(* Logix 5000 project; controller PHOTON Emulate 5570 rev 30.12; software revision 30.00 *)

TASK MainTask (periodic, rate 10000 ms, priority 1, watchdog 10000 ms) : MainProgram

MODULES
   Local : Emulate 5570 (ICP 2, rev 30.12)
       : vendor 1 type 0 code 15 (ICP 0, rev 1.1, Output RPI 50 ms)
END_MODULES

TYPE UDT_BA :
STRUCT
   AL : BOOL[128];
END_STRUCT
END_TYPE

VAR_GLOBAL   (* controller tags *)
   hash_valid : BOOL;
   hash_value : INT[32];
   hash_value_id : DINT;
   open_msg : INT[96];
   open_msg_id : DINT;
   open_msg_valid : BOOL;
   SCAN_CYCLE_TIME : DINT;
END_VAR

PROGRAM MainProgram   (* main routine MainRoutine *)
VAR
   PHT_Bit_indxj : DINT;
   PHT_Byte_indxi : DINT;
   PHT_Ceilmod : DINT;
   PHT_CeilRres : DINT;
   PHT_CompressFunction_BitOffSet : DINT;
   PHT_D : DINT;
   PHT_Digest : DINT[60];
   PHT_DIGESTSIZE : DINT;
   PHT_GetByte_BitOffSet : DINT;
   PHT_GetByte_i : DINT;
   PHT_GetByte_Indx : DINT;
   PHT_GetByte_j : DINT;
   PHT_GetByte_NoOfBits : DINT;
   PHT_GetByte_Res : DINT;
   PHT_hash_index : DINT;
   PHT_i : DINT;
   PHT_index : DINT;
   PHT_Init_i : DINT;
   PHT_isPadding : BOOL;
   PHT_IV : INT[8,8];
   PHT_j : DINT;
   PHT_Message : DINT[1024];
   PHT_MessIndex : DINT;
   PHT_MsgBitLen : DINT;
   PHT_Padded : DINT[1024];
   PHT_Padded_bound : DINT;
   PHT_Padded_Index : DINT;
   PHT_Per_i : DINT;
   PHT_Per_j : DINT;
   PHT_Per_r : DINT;
   PHT_RATE : DINT;
   PHT_RATEP : DINT;
   PHT_RC : DINT[8,12];
   PHT_round : DINT;
   PHT_S : DINT;
   PHT_SCS_c : DINT;
   PHT_SCS_i : DINT;
   PHT_SCS_index : DINT;
   PHT_SCS_indxi : DINT;
   PHT_SCS_j : DINT;
   PHT_SCS_OS : DINT[8,8];
   PHT_SCS_r : DINT;
   PHT_SCS_v : DINT[2];
   PHT_Squeeze_i : DINT;
   PHT_Squeeze_tmp : DINT;
   PHT_State : DINT[8,8];
   PHT_Table : DINT[8,256,2];
   PHT_Tmp : DINT[2];
   PHT_Ver : DINT;
   PHT_WordToByte_BitOffSet : DINT;
   PHT_WordToByte_i : DINT;
   PHT_WordToByte_indxi : DINT;
   PHT_WordToByte_indxj : DINT;
   PHT_WordToByte_j : DINT;
   PHT_WordToByte_NoOfBits : DINT;
   PHT_WordToByte_WordOffset : DINT;
   PHT_WordXorByte_BitOffSet : DINT;
   PHT_WordXorByte_i : DINT;
   PHT_WordXorByte_j : DINT;
   PHT_WordXorByte_NoOfBits : DINT;
   PHT_WordXorByte_Str : DINT[1024];
   PHT_WordXorByte_WordOffset : DINT;
   PHT_WriteByte_BitOffset : DINT;
   PHT_WriteByte_i : DINT;
   PHT_WriteByte_LocalFilter : DINT;
   PHT_WriteByte_NoOfBits : DINT;
   PHT_WriteByte_Value : DINT;
   Test_i : DINT;
END_VAR

ROUTINE MainRoutine   (* ladder *)
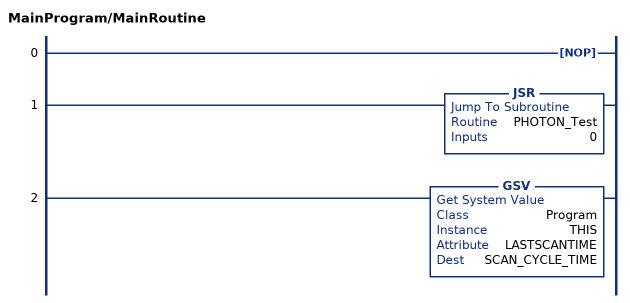
   0: NOP();
   1: JSR(PHOTON_Test,0);
   2: GSV(Program,THIS,LASTSCANTIME,SCAN_CYCLE_TIME);
END_ROUTINE

ROUTINE PHOTON   (* structured text *)
   
   
   JSR(PHOTON_Init);
   
   PHT_isPadding:=0;
   
   PHT_MessIndex:=0;
   while PHT_MessIndex <= PHT_MsgBitLen - PHT_RATE do
   
   	PHT_CompressFunction_BitOffSet:=PHT_MessIndex;
   	JSR(PHOTON_CompressFunction);
   
   	PHT_MessIndex:=PHT_MessIndex + PHT_RATE;
   end_while;
   
   
   PHT_Ceilmod:=PHT_MsgBitLen-PHT_MessIndex;
   PHT_Padded_bound:=PHT_Ceilmod/8;
   PHT_Ceilmod:= PHT_Ceilmod Mod 8;
   if PHT_Ceilmod<>0 then
   	PHT_Padded_bound:=PHT_Padded_bound+1;
   end_if;
   
   
   PHT_hash_index:=PHT_MessIndex/8;
   
   for PHT_i:=0 to PHT_Padded_bound-1 by 1 do
   	PHT_Padded[PHT_i]:=PHT_Message[PHT_hash_index + PHT_i];
   end_for;
   PHT_Padded[PHT_i]:=16#80;
   
   PHT_isPadding:=1;
   
   
   
   PHT_CompressFunction_BitOffSet:=PHT_MessIndex and 16#07;
   JSR(PHOTON_CompressFunction);
   
   
   JSR(PHOTON_Squeeze);
   
END_ROUTINE

ROUTINE PHOTON_CompressFunction   (* structured text *)
   
   PHT_WordXorByte_NoOfBits:=PHT_RATE;
   PHT_WordXorByte_WordOffset:=0;
   PHT_WordXorByte_BitOffSet:= PHT_CompressFunction_BitOffSet;
   
   JSR(PHOTON_WordXorByte);
   
   
   JSR(PHOTON_Permutation);
END_ROUTINE

ROUTINE PHOTON_GetByte   (* structured text *)
   (*byte GetByte(const byte*str, int BitOffSet, int NoOfBits)
       if S==8:
           if (BitOffSet & 0x7):
               res=((str[BitOffSet >> 3] << 4) | (str[(BitOffSet >> 3) + 1] >> 4))
           else:
               res=str[BitOffSet >> 3]
       else:
           res=(str[BitOffSet>>3] >> (4-(BitOffSet&0x4))) & ((1<<S)-1)
   
       return res
   	*)
   
   
   PHT_GetByte_Res:=0;
   
   PHT_GetByte_Indx:=PHT_GetByte_BitOffSet/8;
   
   If PHT_S=8 Then
   	PHT_Tmp[0]:=PHT_GetByte_BitOffSet AND 16#7;
   	if PHT_Tmp[0]<>0 Then
   		If PHT_isPadding Then
   			PHT_Tmp[0]:=PHT_Padded[PHT_GetByte_Indx]*16;
   			PHT_Tmp[1]:=PHT_Padded[PHT_GetByte_Indx+1]/16;
   		else
   			PHT_Tmp[0]:=PHT_Message[PHT_GetByte_Indx]*16;
   			PHT_Tmp[1]:=PHT_Message[PHT_GetByte_Indx+1]/16;
   		End_If;
   		PHT_GetByte_Res:=(PHT_Tmp[0] OR PHT_Tmp[1]) AND 16#FF;
   	else
   		If PHT_isPadding Then
   			PHT_GetByte_Res:=PHT_Padded[PHT_GetByte_Indx];
   		Else
   			PHT_GetByte_Res:=PHT_Message[PHT_GetByte_Indx];
   		End_If;
   	End_if;
   Else
   	If PHT_isPadding Then
   		PHT_Tmp[0]:=PHT_Padded[PHT_GetByte_Indx];
   	Else
   		PHT_Tmp[0]:=PHT_Message[PHT_GetByte_Indx];
   	End_If;
   
   
   	PHT_Tmp[1]:=4-(PHT_GetByte_BitOffSet AND 16#4);
   	Case PHT_Tmp[1] OF
   		1:
   			PHT_Tmp[0]:=PHT_Tmp[0]/2;
   		2:
   			PHT_Tmp[0]:=PHT_Tmp[0]/4;
   		3:
   			PHT_Tmp[0]:=PHT_Tmp[0]/8;
   		4:
   			PHT_Tmp[0]:=PHT_Tmp[0]/16;
   	End_CASE;
   	PHT_GetByte_Res:=PHT_Tmp[0] & 16#f;
   
   End_if;
   
   
END_ROUTINE

ROUTINE PHOTON_Init   (* structured text *)
   PHT_round:=12; // 12
   if PHT_Ver >= 5 then
   	PHT_S:= 8;
   else
   	PHT_S:=4;
   end_if;
   
   CASE PHT_Ver OF
   	 0:
   		PHT_D:=5;
   		PHT_S:=4;
   		PHT_RATE:=20;
   		PHT_RATEP:=16;
   		PHT_DIGESTSIZE:=80;
   		 PHT_RC[0,0]:=1;
   		 PHT_RC[0,1]:=3;
   		 PHT_RC[0,2]:=7;
   		 PHT_RC[0,3]:=14;
   		 PHT_RC[0,4]:=13;
   		 PHT_RC[0,5]:=11;
   		 PHT_RC[0,6]:=6;
   		 PHT_RC[0,7]:=12;
   		 PHT_RC[0,8]:=9;
   		 PHT_RC[0,9]:=2;
   		 PHT_RC[0,10]:=5;
   		 PHT_RC[0,11]:=10;
   		 PHT_RC[1,0]:=0;
   		 PHT_RC[1,1]:=2;
   		 PHT_RC[1,2]:=6;
   		 PHT_RC[1,3]:=15;
   		 PHT_RC[1,4]:=12;
   		 PHT_RC[1,5]:=10;
   		 PHT_RC[1,6]:=7;
   		 PHT_RC[1,7]:=13;
   		 PHT_RC[1,8]:=8;
   		 PHT_RC[1,9]:=3;
   		 PHT_RC[1,10]:=4;
   		 PHT_RC[1,11]:=11;
   		 PHT_RC[2,0]:=2;
   		 PHT_RC[2,1]:=0;
   		 PHT_RC[2,2]:=4;
   		 PHT_RC[2,3]:=13;
   		 PHT_RC[2,4]:=14;
   		 PHT_RC[2,5]:=8;
   		 PHT_RC[2,6]:=5;
   		 PHT_RC[2,7]:=15;
   		 PHT_RC[2,8]:=10;
   		 PHT_RC[2,9]:=1;
   		 PHT_RC[2,10]:=6;
   		 PHT_RC[2,11]:=9;
   		 PHT_RC[3,0]:=7;
   		 PHT_RC[3,1]:=5;
   		 PHT_RC[3,2]:=1;
   		 PHT_RC[3,3]:=8;
   		 PHT_RC[3,4]:=11;
   		 PHT_RC[3,5]:=13;
   		 PHT_RC[3,6]:=0;
   		 PHT_RC[3,7]:=10;
   		 PHT_RC[3,8]:=15;
   		 PHT_RC[3,9]:=4;
   		 PHT_RC[3,10]:=3;
   		 PHT_RC[3,11]:=12;
   		 PHT_RC[4,0]:=5;
   		 PHT_RC[4,1]:=7;
   		 PHT_RC[4,2]:=3;
   		 PHT_RC[4,3]:=10;
   		 PHT_RC[4,4]:=9;
   		 PHT_RC[4,5]:=15;
   		 PHT_RC[4,6]:=2;
   		 PHT_RC[4,7]:=8;
   		 PHT_RC[4,8]:=13;
   		 PHT_RC[4,9]:=6;
   		 PHT_RC[4,10]:=1;
   		 PHT_RC[4,11]:=14;
   		 PHT_State[0,0]:=0;
   		 PHT_State[0,1]:=0;
   		 PHT_State[0,2]:=0;
   		 PHT_State[0,3]:=0;
   		 PHT_State[0,4]:=0;
   		 PHT_State[1,0]:=0;
   		 PHT_State[1,1]:=0;
   		 PHT_State[1,2]:=0;
   		 PHT_State[1,3]:=0;
   		 PHT_State[1,4]:=0;
   		 PHT_State[2,0]:=0;
   		 PHT_State[2,1]:=0;
   		 PHT_State[2,2]:=0;
   		 PHT_State[2,3]:=0;
   		 PHT_State[2,4]:=0;
   		 PHT_State[3,0]:=0;
   		 PHT_State[3,1]:=0;
   		 PHT_State[3,2]:=0;
   		 PHT_State[3,3]:=0;
   		 PHT_State[3,4]:=1;
   		 PHT_State[4,0]:=4;
   		 PHT_State[4,1]:=1;
   		 PHT_State[4,2]:=4;
   		 PHT_State[4,3]:=1;
   		 PHT_State[4,4]:=0;
   		 PHT_Table[0,0,0]:=832452;
   		 PHT_Table[1,0,0]:=761220;
   		 PHT_Table[2,0,0]:=422330;
   		 PHT_Table[3,0,0]:=438137;
   		 PHT_Table[4,0,0]:=736335;
   		 PHT_Table[0,1,0]:=371795;
   		 PHT_Table[1,1,0]:=663907;
   		 PHT_Table[2,1,0]:=783534;
   		 PHT_Table[3,1,0]:=780786;
   		 PHT_Table[4,1,0]:=705849;
   		 PHT_Table[0,2,0]:=444514;
   		 PHT_Table[1,2,0]:=843586;
   		 PHT_Table[2,2,0]:=240069;
   		 PHT_Table[3,2,0]:=220845;
   		 PHT_Table[4,2,0]:=820782;
   		 PHT_Table[0,3,0]:=743096;
   		 PHT_Table[1,3,0]:=334136;
   		 PHT_Table[2,3,0]:=844375;
   		 PHT_Table[3,3,0]:=818657;
   		 PHT_Table[4,3,0]:=355213;
   		 PHT_Table[0,4,0]:=597911;
   		 PHT_Table[1,4,0]:=113895;
   		 PHT_Table[2,4,0]:=886036;
   		 PHT_Table[3,4,0]:=870027;
   		 PHT_Table[4,4,0]:=129398;
   		 PHT_Table[0,5,0]:=0;
   		 PHT_Table[1,5,0]:=0;
   		 PHT_Table[2,5,0]:=0;
   		 PHT_Table[3,5,0]:=0;
   		 PHT_Table[4,5,0]:=0;
   		 PHT_Table[0,6,0]:=687014;
   		 PHT_Table[1,6,0]:=475846;
   		 PHT_Table[2,6,0]:=383103;
   		 PHT_Table[3,6,0]:=389588;
   		 PHT_Table[4,6,0]:=506465;
   		 PHT_Table[0,7,0]:=892634;
   		 PHT_Table[1,7,0]:=640634;
   		 PHT_Table[2,7,0]:=1002386;
   		 PHT_Table[3,7,0]:=992076;
   		 PHT_Table[4,7,0]:=650659;
   		 PHT_Table[0,8,0]:=222257;
   		 PHT_Table[1,8,0]:=458273;
   		 PHT_Table[2,8,0]:=548203;
   		 PHT_Table[3,8,0]:=571231;
   		 PHT_Table[4,8,0]:=410391;
   		 PHT_Table[0,9,0]:=981739;
   		 PHT_Table[1,9,0]:=997467;
   		 PHT_Table[2,9,0]:=464633;
   		 PHT_Table[3,9,0]:=496659;
   		 PHT_Table[4,9,0]:=1027764;
   		 PHT_Table[0,10,0]:=1038325;
   		 PHT_Table[1,10,0]:=877477;
   		 PHT_Table[2,10,0]:=928977;
   		 PHT_Table[3,10,0]:=923686;
   		 PHT_Table[4,10,0]:=884568;
   		 PHT_Table[0,11,0]:=537225;
   		 PHT_Table[1,11,0]:=255769;
   		 PHT_Table[2,11,0]:=311100;
   		 PHT_Table[3,11,0]:=314046;
   		 PHT_Table[4,11,0]:=207002;
   		 PHT_Table[0,12,0]:=295245;
   		 PHT_Table[1,12,0]:=555677;
   		 PHT_Table[2,12,0]:=183942;
   		 PHT_Table[3,12,0]:=157127;
   		 PHT_Table[4,12,0]:=529621;
   		 PHT_Table[0,13,0]:=517500;
   		 PHT_Table[1,13,0]:=951484;
   		 PHT_Table[2,13,0]:=693229;
   		 PHT_Table[3,13,0]:=709272;
   		 PHT_Table[4,13,0]:=939970;
   		 PHT_Table[0,14,0]:=77086;
   		 PHT_Table[1,14,0]:=154622;
   		 PHT_Table[2,14,0]:=604712;
   		 PHT_Table[3,14,0]:=625717;
   		 PHT_Table[4,14,0]:=184812;
   		 PHT_Table[0,15,0]:=149807;
   		 PHT_Table[1,15,0]:=304607;
   		 PHT_Table[2,15,0]:=91971;
   		 PHT_Table[3,15,0]:=80746;
   		 PHT_Table[4,15,0]:=299771;
   	 1:
   		PHT_D:=6;
   		PHT_S:=4;
   		PHT_RATE:=16;
   		PHT_RATEP:=16;
   		PHT_DIGESTSIZE:=128;
   		 PHT_RC[0,0]:=1;
   		 PHT_RC[0,1]:=3;
   		 PHT_RC[0,2]:=7;
   		 PHT_RC[0,3]:=14;
   		 PHT_RC[0,4]:=13;
   		 PHT_RC[0,5]:=11;
   		 PHT_RC[0,6]:=6;
   		 PHT_RC[0,7]:=12;
   		 PHT_RC[0,8]:=9;
   		 PHT_RC[0,9]:=2;
   		 PHT_RC[0,10]:=5;
   		 PHT_RC[0,11]:=10;
   		 PHT_RC[1,0]:=0;
   		 PHT_RC[1,1]:=2;
   		 PHT_RC[1,2]:=6;
   		 PHT_RC[1,3]:=15;
   		 PHT_RC[1,4]:=12;
   		 PHT_RC[1,5]:=10;
   		 PHT_RC[1,6]:=7;
   		 PHT_RC[1,7]:=13;
   		 PHT_RC[1,8]:=8;
   		 PHT_RC[1,9]:=3;
   		 PHT_RC[1,10]:=4;
   		 PHT_RC[1,11]:=11;
   		 PHT_RC[2,0]:=2;
   		 PHT_RC[2,1]:=0;
   		 PHT_RC[2,2]:=4;
   		 PHT_RC[2,3]:=13;
   		 PHT_RC[2,4]:=14;
   		 PHT_RC[2,5]:=8;
   		 PHT_RC[2,6]:=5;
   		 PHT_RC[2,7]:=15;
   		 PHT_RC[2,8]:=10;
   		 PHT_RC[2,9]:=1;
   		 PHT_RC[2,10]:=6;
   		 PHT_RC[2,11]:=9;
   		 PHT_RC[3,0]:=6;
   		 PHT_RC[3,1]:=4;
   		 PHT_RC[3,2]:=0;
   		 PHT_RC[3,3]:=9;
   		 PHT_RC[3,4]:=10;
   		 PHT_RC[3,5]:=12;
   		 PHT_RC[3,6]:=1;
   		 PHT_RC[3,7]:=11;
   		 PHT_RC[3,8]:=14;
   		 PHT_RC[3,9]:=5;
   		 PHT_RC[3,10]:=2;
   		 PHT_RC[3,11]:=13;
   		 PHT_RC[4,0]:=7;
   		 PHT_RC[4,1]:=5;
   		 PHT_RC[4,2]:=1;
   		 PHT_RC[4,3]:=8;
   		 PHT_RC[4,4]:=11;
   		 PHT_RC[4,5]:=13;
   		 PHT_RC[4,6]:=0;
   		 PHT_RC[4,7]:=10;
   		 PHT_RC[4,8]:=15;
   		 PHT_RC[4,9]:=4;
   		 PHT_RC[4,10]:=3;
   		 PHT_RC[4,11]:=12;
   		 PHT_RC[5,0]:=5;
   		 PHT_RC[5,1]:=7;
   		 PHT_RC[5,2]:=3;
   		 PHT_RC[5,3]:=10;
   		 PHT_RC[5,4]:=9;
   		 PHT_RC[5,5]:=15;
   		 PHT_RC[5,6]:=2;
   		 PHT_RC[5,7]:=8;
   		 PHT_RC[5,8]:=13;
   		 PHT_RC[5,9]:=6;
   		 PHT_RC[5,10]:=1;
   		 PHT_RC[5,11]:=14;
   		 PHT_State[0,0]:=0;
   		 PHT_State[0,1]:=0;
   		 PHT_State[0,2]:=0;
   		 PHT_State[0,3]:=0;
   		 PHT_State[0,4]:=0;
   		 PHT_State[0,5]:=0;
   		 PHT_State[1,0]:=0;
   		 PHT_State[1,1]:=0;
   		 PHT_State[1,2]:=0;
   		 PHT_State[1,3]:=0;
   		 PHT_State[1,4]:=0;
   		 PHT_State[1,5]:=0;
   		 PHT_State[2,0]:=0;
   		 PHT_State[2,1]:=0;
   		 PHT_State[2,2]:=0;
   		 PHT_State[2,3]:=0;
   		 PHT_State[2,4]:=0;
   		 PHT_State[2,5]:=0;
   		 PHT_State[3,0]:=0;
   		 PHT_State[3,1]:=0;
   		 PHT_State[3,2]:=0;
   		 PHT_State[3,3]:=0;
   		 PHT_State[3,4]:=0;
   		 PHT_State[3,5]:=0;
   		 PHT_State[4,0]:=0;
   		 PHT_State[4,1]:=0;
   		 PHT_State[4,2]:=0;
   		 PHT_State[4,3]:=0;
   		 PHT_State[4,4]:=0;
   		 PHT_State[4,5]:=0;
   		 PHT_State[5,0]:=2;
   		 PHT_State[5,1]:=0;
   		 PHT_State[5,2]:=1;
   		 PHT_State[5,3]:=0;
   		 PHT_State[5,4]:=1;
   		 PHT_State[5,5]:=0;
   		 PHT_Table[0,0,0]:=13366218;
   		 PHT_Table[1,0,0]:=12151179;
   		 PHT_Table[2,0,0]:=11308343;
   		 PHT_Table[3,0,0]:=10200903;
   		 PHT_Table[4,0,0]:=11444699;
   		 PHT_Table[5,0,0]:=12532906;
   		 PHT_Table[0,1,0]:=5938270;
   		 PHT_Table[1,1,0]:=10662506;
   		 PHT_Table[2,1,0]:=15032783;
   		 PHT_Table[3,1,0]:=2813759;
   		 PHT_Table[4,1,0]:=15590426;
   		 PHT_Table[5,1,0]:=11126254;
   		 PHT_Table[0,2,0]:=7137381;
   		 PHT_Table[1,2,0]:=13450572;
   		 PHT_Table[2,2,0]:=5656458;
   		 PHT_Table[3,2,0]:=14441002;
   		 PHT_Table[4,2,0]:=5724668;
   		 PHT_Table[5,2,0]:=13534805;
   		 PHT_Table[0,3,0]:=11916983;
   		 PHT_Table[1,3,0]:=5357877;
   		 PHT_Table[2,3,0]:=8075630;
   		 PHT_Table[3,3,0]:=1408654;
   		 PHT_Table[4,3,0]:=8352405;
   		 PHT_Table[5,3,0]:=6122359;
   		 PHT_Table[0,4,0]:=9531284;
   		 PHT_Table[1,4,0]:=1825761;
   		 PHT_Table[2,4,0]:=4844792;
   		 PHT_Table[3,4,0]:=11618424;
   		 PHT_Table[4,4,0]:=4408769;
   		 PHT_Table[5,4,0]:=1505604;
   		 PHT_Table[0,5,0]:=0;
   		 PHT_Table[1,5,0]:=0;
   		 PHT_Table[2,5,0]:=0;
   		 PHT_Table[3,5,0]:=0;
   		 PHT_Table[4,5,0]:=0;
   		 PHT_Table[5,5,0]:=0;
   		 PHT_Table[0,6,0]:=10951599;
   		 PHT_Table[1,6,0]:=7623879;
   		 PHT_Table[2,6,0]:=16433853;
   		 PHT_Table[3,6,0]:=4717933;
   		 PHT_Table[4,6,0]:=16381991;
   		 PHT_Table[5,6,0]:=7453439;
   		 PHT_Table[0,7,0]:=14237394;
   		 PHT_Table[1,7,0]:=10288249;
   		 PHT_Table[2,7,0]:=2979556;
   		 PHT_Table[3,7,0]:=13182116;
   		 PHT_Table[4,7,0]:=2632553;
   		 PHT_Table[5,7,0]:=9694498;
   		 PHT_Table[0,8,0]:=3568699;
   		 PHT_Table[1,8,0]:=7311142;
   		 PHT_Table[2,8,0]:=11742789;
   		 PHT_Table[3,8,0]:=16168213;
   		 PHT_Table[4,8,0]:=12238310;
   		 PHT_Table[5,8,0]:=6767547;
   		 PHT_Table[0,9,0]:=15682281;
   		 PHT_Table[1,9,0]:=15954783;
   		 PHT_Table[2,9,0]:=10377377;
   		 PHT_Table[3,9,0]:=4166065;
   		 PHT_Table[4,9,0]:=9606799;
   		 PHT_Table[5,9,0]:=16035481;
   		 PHT_Table[0,10,0]:=16615409;
   		 PHT_Table[1,10,0]:=14083757;
   		 PHT_Table[2,10,0]:=2073458;
   		 PHT_Table[3,10,0]:=7148114;
   		 PHT_Table[4,10,0]:=1317949;
   		 PHT_Table[5,10,0]:=14188305;
   		 PHT_Table[0,11,0]:=8626828;
   		 PHT_Table[1,11,0]:=4083219;
   		 PHT_Table[2,11,0]:=13113131;
   		 PHT_Table[3,11,0]:=14928795;
   		 PHT_Table[4,11,0]:=12963699;
   		 PHT_Table[5,11,0]:=3811532;
   		 PHT_Table[0,12,0]:=4739398;
   		 PHT_Table[1,12,0]:=8857496;
   		 PHT_Table[2,12,0]:=6593052;
   		 PHT_Table[3,12,0]:=7892188;
   		 PHT_Table[4,12,0]:=7040680;
   		 PHT_Table[5,12,0]:=8721510;
   		 PHT_Table[0,13,0]:=8267133;
   		 PHT_Table[1,13,0]:=15247550;
   		 PHT_Table[2,13,0]:=14136409;
   		 PHT_Table[3,13,0]:=9361865;
   		 PHT_Table[4,13,0]:=13751118;
   		 PHT_Table[5,13,0]:=14833629;
   		 PHT_Table[0,14,0]:=1232152;
   		 PHT_Table[1,14,0]:=2463218;
   		 PHT_Table[2,14,0]:=8518611;
   		 PHT_Table[3,14,0]:=5407715;
   		 PHT_Table[4,14,0]:=8817330;
   		 PHT_Table[5,14,0]:=2937224;
   		 PHT_Table[0,15,0]:=2406691;
   		 PHT_Table[1,15,0]:=4856532;
   		 PHT_Table[2,15,0]:=3331478;
   		 PHT_Table[3,15,0]:=10761974;
   		 PHT_Table[4,15,0]:=3946324;
   		 PHT_Table[5,15,0]:=4952627;
   	 2:
   		PHT_D:=7;
   		PHT_S:=4;
   		PHT_RATE:=36;
   		PHT_RATEP:=36;
   		PHT_DIGESTSIZE:=160;
   		 PHT_RC[0,0]:=1;
   		 PHT_RC[0,1]:=3;
   		 PHT_RC[0,2]:=7;
   		 PHT_RC[0,3]:=14;
   		 PHT_RC[0,4]:=13;
   		 PHT_RC[0,5]:=11;
   		 PHT_RC[0,6]:=6;
   		 PHT_RC[0,7]:=12;
   		 PHT_RC[0,8]:=9;
   		 PHT_RC[0,9]:=2;
   		 PHT_RC[0,10]:=5;
   		 PHT_RC[0,11]:=10;
   		 PHT_RC[1,0]:=0;
   		 PHT_RC[1,1]:=2;
   		 PHT_RC[1,2]:=6;
   		 PHT_RC[1,3]:=15;
   		 PHT_RC[1,4]:=12;
   		 PHT_RC[1,5]:=10;
   		 PHT_RC[1,6]:=7;
   		 PHT_RC[1,7]:=13;
   		 PHT_RC[1,8]:=8;
   		 PHT_RC[1,9]:=3;
   		 PHT_RC[1,10]:=4;
   		 PHT_RC[1,11]:=11;
   		 PHT_RC[2,0]:=3;
   		 PHT_RC[2,1]:=1;
   		 PHT_RC[2,2]:=5;
   		 PHT_RC[2,3]:=12;
   		 PHT_RC[2,4]:=15;
   		 PHT_RC[2,5]:=9;
   		 PHT_RC[2,6]:=4;
   		 PHT_RC[2,7]:=14;
   		 PHT_RC[2,8]:=11;
   		 PHT_RC[2,9]:=0;
   		 PHT_RC[2,10]:=7;
   		 PHT_RC[2,11]:=8;
   		 PHT_RC[3,0]:=4;
   		 PHT_RC[3,1]:=6;
   		 PHT_RC[3,2]:=2;
   		 PHT_RC[3,3]:=11;
   		 PHT_RC[3,4]:=8;
   		 PHT_RC[3,5]:=14;
   		 PHT_RC[3,6]:=3;
   		 PHT_RC[3,7]:=9;
   		 PHT_RC[3,8]:=12;
   		 PHT_RC[3,9]:=7;
   		 PHT_RC[3,10]:=0;
   		 PHT_RC[3,11]:=15;
   		 PHT_RC[4,0]:=2;
   		 PHT_RC[4,1]:=0;
   		 PHT_RC[4,2]:=4;
   		 PHT_RC[4,3]:=13;
   		 PHT_RC[4,4]:=14;
   		 PHT_RC[4,5]:=8;
   		 PHT_RC[4,6]:=5;
   		 PHT_RC[4,7]:=15;
   		 PHT_RC[4,8]:=10;
   		 PHT_RC[4,9]:=1;
   		 PHT_RC[4,10]:=6;
   		 PHT_RC[4,11]:=9;
   		 PHT_RC[5,0]:=7;
   		 PHT_RC[5,1]:=5;
   		 PHT_RC[5,2]:=1;
   		 PHT_RC[5,3]:=8;
   		 PHT_RC[5,4]:=11;
   		 PHT_RC[5,5]:=13;
   		 PHT_RC[5,6]:=0;
   		 PHT_RC[5,7]:=10;
   		 PHT_RC[5,8]:=15;
   		 PHT_RC[5,9]:=4;
   		 PHT_RC[5,10]:=3;
   		 PHT_RC[5,11]:=12;
   		 PHT_RC[6,0]:=5;
   		 PHT_RC[6,1]:=7;
   		 PHT_RC[6,2]:=3;
   		 PHT_RC[6,3]:=10;
   		 PHT_RC[6,4]:=9;
   		 PHT_RC[6,5]:=15;
   		 PHT_RC[6,6]:=2;
   		 PHT_RC[6,7]:=8;
   		 PHT_RC[6,8]:=13;
   		 PHT_RC[6,9]:=6;
   		 PHT_RC[6,10]:=1;
   		 PHT_RC[6,11]:=14;
   		 PHT_State[0,0]:=0;
   		 PHT_State[0,1]:=0;
   		 PHT_State[0,2]:=0;
   		 PHT_State[0,3]:=0;
   		 PHT_State[0,4]:=0;
   		 PHT_State[0,5]:=0;
   		 PHT_State[0,6]:=0;
   		 PHT_State[1,0]:=0;
   		 PHT_State[1,1]:=0;
   		 PHT_State[1,2]:=0;
   		 PHT_State[1,3]:=0;
   		 PHT_State[1,4]:=0;
   		 PHT_State[1,5]:=0;
   		 PHT_State[1,6]:=0;
   		 PHT_State[2,0]:=0;
   		 PHT_State[2,1]:=0;
   		 PHT_State[2,2]:=0;
   		 PHT_State[2,3]:=0;
   		 PHT_State[2,4]:=0;
   		 PHT_State[2,5]:=0;
   		 PHT_State[2,6]:=0;
   		 PHT_State[3,0]:=0;
   		 PHT_State[3,1]:=0;
   		 PHT_State[3,2]:=0;
   		 PHT_State[3,3]:=0;
   		 PHT_State[3,4]:=0;
   		 PHT_State[3,5]:=0;
   		 PHT_State[3,6]:=0;
   		 PHT_State[4,0]:=0;
   		 PHT_State[4,1]:=0;
   		 PHT_State[4,2]:=0;
   		 PHT_State[4,3]:=0;
   		 PHT_State[4,4]:=0;
   		 PHT_State[4,5]:=0;
   		 PHT_State[4,6]:=0;
   		 PHT_State[5,0]:=0;
   		 PHT_State[5,1]:=0;
   		 PHT_State[5,2]:=0;
   		 PHT_State[5,3]:=0;
   		 PHT_State[5,4]:=0;
   		 PHT_State[5,5]:=0;
   		 PHT_State[5,6]:=0;
   		 PHT_State[6,0]:=0;
   		 PHT_State[6,1]:=2;
   		 PHT_State[6,2]:=8;
   		 PHT_State[6,3]:=2;
   		 PHT_State[6,4]:=4;
   		 PHT_State[6,5]:=2;
   		 PHT_State[6,6]:=4;
   		 PHT_Table[0,0,0]:=207173177;
   		 PHT_Table[1,0,0]:=95901857;
   		 PHT_Table[2,0,0]:=243847721;
   		 PHT_Table[3,0,0]:=212974363;
   		 PHT_Table[4,0,0]:=210906504;
   		 PHT_Table[5,0,0]:=236619131;
   		 PHT_Table[6,0,0]:=93545365;
   		 PHT_Table[0,1,0]:=91409346;
   		 PHT_Table[1,1,0]:=128939748;
   		 PHT_Table[2,1,0]:=224794754;
   		 PHT_Table[3,1,0]:=94677578;
   		 PHT_Table[4,1,0]:=86540646;
   		 PHT_Table[5,1,0]:=223242234;
   		 PHT_Table[6,1,0]:=120372263;
   		 PHT_Table[0,2,0]:=113083277;
   		 PHT_Table[1,2,0]:=197833817;
   		 PHT_Table[2,2,0]:=121958685;
   		 PHT_Table[3,2,0]:=113888412;
   		 PHT_Table[4,2,0]:=114368324;
   		 PHT_Table[5,2,0]:=127224748;
   		 PHT_Table[6,2,0]:=198719707;
   		 PHT_Table[0,3,0]:=195128417;
   		 PHT_Table[1,3,0]:=173974386;
   		 PHT_Table[2,3,0]:=255038529;
   		 PHT_Table[3,3,0]:=189945125;
   		 PHT_Table[4,3,0]:=185878835;
   		 PHT_Table[5,3,0]:=254229221;
   		 PHT_Table[6,3,0]:=169264666;
   		 PHT_Table[0,4,0]:=153878011;
   		 PHT_Table[1,4,0]:=35139141;
   		 PHT_Table[2,4,0]:=65981099;
   		 PHT_Table[3,4,0]:=152375633;
   		 PHT_Table[4,4,0]:=163228910;
   		 PHT_Table[5,4,0]:=55894657;
   		 PHT_Table[6,4,0]:=46129074;
   		 PHT_Table[0,5,0]:=0;
   		 PHT_Table[1,5,0]:=0;
   		 PHT_Table[2,5,0]:=0;
   		 PHT_Table[3,5,0]:=0;
   		 PHT_Table[4,5,0]:=0;
   		 PHT_Table[5,5,0]:=0;
   		 PHT_Table[6,5,0]:=0;
   		 PHT_Table[0,6,0]:=182760884;
   		 PHT_Table[1,6,0]:=243133688;
   		 PHT_Table[2,6,0]:=164373300;
   		 PHT_Table[3,6,0]:=175667079;
   		 PHT_Table[4,6,0]:=172176076;
   		 PHT_Table[5,6,0]:=160419543;
   		 PHT_Table[6,6,0]:=239819598;
   		 PHT_Table[0,7,0]:=220000236;
   		 PHT_Table[1,7,0]:=26482475;
   		 PHT_Table[2,7,0]:=142042460;
   		 PHT_Table[3,7,0]:=228301241;
   		 PHT_Table[4,7,0]:=231036535;
   		 PHT_Table[5,7,0]:=145912137;
   		 PHT_Table[6,7,0]:=30342849;
   		 PHT_Table[0,8,0]:=63916111;
   		 PHT_Table[1,8,0]:=207995581;
   		 PHT_Table[2,8,0]:=170060191;
   		 PHT_Table[3,8,0]:=57501398;
   		 PHT_Table[4,8,0]:=66690594;
   		 PHT_Table[5,8,0]:=182135894;
   		 PHT_Table[6,8,0]:=217351420;
   		 PHT_Table[0,9,0]:=248752035;
   		 PHT_Table[1,9,0]:=233952662;
   		 PHT_Table[2,9,0]:=39161027;
   		 PHT_Table[3,9,0]:=251068271;
   		 PHT_Table[4,9,0]:=238864469;
   		 PHT_Table[5,9,0]:=40459551;
   		 PHT_Table[6,9,0]:=221936189;
   		 PHT_Table[0,10,0]:=261521014;
   		 PHT_Table[1,10,0]:=164796956;
   		 PHT_Table[2,10,0]:=78265270;
   		 PHT_Table[3,10,0]:=266132941;
   		 PHT_Table[4,10,0]:=258716586;
   		 PHT_Table[5,10,0]:=79800621;
   		 PHT_Table[6,10,0]:=157804393;
   		 PHT_Table[0,11,0]:=141435950;
   		 PHT_Table[1,11,0]:=104554959;
   		 PHT_Table[2,11,0]:=85032414;
   		 PHT_Table[3,11,0]:=138359795;
   		 PHT_Table[4,11,0]:=149804817;
   		 PHT_Table[5,11,0]:=100406963;
   		 PHT_Table[6,11,0]:=115491558;
   		 PHT_Table[0,12,0]:=70717975;
   		 PHT_Table[1,12,0]:=59521390;
   		 PHT_Table[2,12,0]:=194621431;
   		 PHT_Table[3,12,0]:=76450024;
   		 PHT_Table[4,12,0]:=75496089;
   		 PHT_Table[5,12,0]:=199660488;
   		 PHT_Table[6,12,0]:=57745779;
   		 PHT_Table[0,13,0]:=133716568;
   		 PHT_Table[1,13,0]:=266992595;
   		 PHT_Table[2,13,0]:=29050472;
   		 PHT_Table[3,13,0]:=132378174;
   		 PHT_Table[4,13,0]:=126248123;
   		 PHT_Table[5,13,0]:=20823966;
   		 PHT_Table[6,13,0]:=260416911;
   		 PHT_Table[0,14,0]:=21354965;
   		 PHT_Table[1,14,0]:=69422986;
   		 PHT_Table[2,14,0]:=117421941;
   		 PHT_Table[3,14,0]:=19538594;
   		 PHT_Table[4,14,0]:=22510591;
   		 PHT_Table[5,14,0]:=111735858;
   		 PHT_Table[6,14,0]:=73243988;
   		 PHT_Table[0,15,0]:=42635674;
   		 PHT_Table[1,15,0]:=138841399;
   		 PHT_Table[2,15,0]:=215834346;
   		 PHT_Table[3,15,0]:=38225012;
   		 PHT_Table[4,15,0]:=45016541;
   		 PHT_Table[5,15,0]:=208918628;
   		 PHT_Table[6,15,0]:=145299880;
   	 3:
   		PHT_D:=7;
   		PHT_S:=4;
   		PHT_RATE:=4;
   		PHT_RATEP:=4;
   		PHT_DIGESTSIZE:=192;
   		 PHT_RC[0,0]:=1;
   		 PHT_RC[0,1]:=3;
   		 PHT_RC[0,2]:=7;
   		 PHT_RC[0,3]:=14;
   		 PHT_RC[0,4]:=13;
   		 PHT_RC[0,5]:=11;
   		 PHT_RC[0,6]:=6;
   		 PHT_RC[0,7]:=12;
   		 PHT_RC[0,8]:=9;
   		 PHT_RC[0,9]:=2;
   		 PHT_RC[0,10]:=5;
   		 PHT_RC[0,11]:=10;
   		 PHT_RC[1,0]:=0;
   		 PHT_RC[1,1]:=2;
   		 PHT_RC[1,2]:=6;
   		 PHT_RC[1,3]:=15;
   		 PHT_RC[1,4]:=12;
   		 PHT_RC[1,5]:=10;
   		 PHT_RC[1,6]:=7;
   		 PHT_RC[1,7]:=13;
   		 PHT_RC[1,8]:=8;
   		 PHT_RC[1,9]:=3;
   		 PHT_RC[1,10]:=4;
   		 PHT_RC[1,11]:=11;
   		 PHT_RC[2,0]:=3;
   		 PHT_RC[2,1]:=1;
   		 PHT_RC[2,2]:=5;
   		 PHT_RC[2,3]:=12;
   		 PHT_RC[2,4]:=15;
   		 PHT_RC[2,5]:=9;
   		 PHT_RC[2,6]:=4;
   		 PHT_RC[2,7]:=14;
   		 PHT_RC[2,8]:=11;
   		 PHT_RC[2,9]:=0;
   		 PHT_RC[2,10]:=7;
   		 PHT_RC[2,11]:=8;
   		 PHT_RC[3,0]:=4;
   		 PHT_RC[3,1]:=6;
   		 PHT_RC[3,2]:=2;
   		 PHT_RC[3,3]:=11;
   		 PHT_RC[3,4]:=8;
   		 PHT_RC[3,5]:=14;
   		 PHT_RC[3,6]:=3;
   		 PHT_RC[3,7]:=9;
   		 PHT_RC[3,8]:=12;
   		 PHT_RC[3,9]:=7;
   		 PHT_RC[3,10]:=0;
   		 PHT_RC[3,11]:=15;
   		 PHT_RC[4,0]:=2;
   		 PHT_RC[4,1]:=0;
   		 PHT_RC[4,2]:=4;
   		 PHT_RC[4,3]:=13;
   		 PHT_RC[4,4]:=14;
   		 PHT_RC[4,5]:=8;
   		 PHT_RC[4,6]:=5;
   		 PHT_RC[4,7]:=15;
   		 PHT_RC[4,8]:=10;
   		 PHT_RC[4,9]:=1;
   		 PHT_RC[4,10]:=6;
   		 PHT_RC[4,11]:=9;
   		 PHT_RC[5,0]:=7;
   		 PHT_RC[5,1]:=5;
   		 PHT_RC[5,2]:=1;
   		 PHT_RC[5,3]:=8;
   		 PHT_RC[5,4]:=11;
   		 PHT_RC[5,5]:=13;
   		 PHT_RC[5,6]:=0;
   		 PHT_RC[5,7]:=10;
   		 PHT_RC[5,8]:=15;
   		 PHT_RC[5,9]:=4;
   		 PHT_RC[5,10]:=3;
   		 PHT_RC[5,11]:=12;
   		 PHT_RC[6,0]:=5;
   		 PHT_RC[6,1]:=7;
   		 PHT_RC[6,2]:=3;
   		 PHT_RC[6,3]:=10;
   		 PHT_RC[6,4]:=9;
   		 PHT_RC[6,5]:=15;
   		 PHT_RC[6,6]:=2;
   		 PHT_RC[6,7]:=8;
   		 PHT_RC[6,8]:=13;
   		 PHT_RC[6,9]:=6;
   		 PHT_RC[6,10]:=1;
   		 PHT_RC[6,11]:=14;
   		 PHT_State[0,0]:=0;
   		 PHT_State[0,1]:=0;
   		 PHT_State[0,2]:=0;
   		 PHT_State[0,3]:=0;
   		 PHT_State[0,4]:=0;
   		 PHT_State[0,5]:=0;
   		 PHT_State[0,6]:=0;
   		 PHT_State[1,0]:=0;
   		 PHT_State[1,1]:=0;
   		 PHT_State[1,2]:=0;
   		 PHT_State[1,3]:=0;
   		 PHT_State[1,4]:=0;
   		 PHT_State[1,5]:=0;
   		 PHT_State[1,6]:=0;
   		 PHT_State[2,0]:=0;
   		 PHT_State[2,1]:=0;
   		 PHT_State[2,2]:=0;
   		 PHT_State[2,3]:=0;
   		 PHT_State[2,4]:=0;
   		 PHT_State[2,5]:=0;
   		 PHT_State[2,6]:=0;
   		 PHT_State[3,0]:=0;
   		 PHT_State[3,1]:=0;
   		 PHT_State[3,2]:=0;
   		 PHT_State[3,3]:=0;
   		 PHT_State[3,4]:=0;
   		 PHT_State[3,5]:=0;
   		 PHT_State[3,6]:=0;
   		 PHT_State[4,0]:=0;
   		 PHT_State[4,1]:=0;
   		 PHT_State[4,2]:=0;
   		 PHT_State[4,3]:=0;
   		 PHT_State[4,4]:=0;
   		 PHT_State[4,5]:=0;
   		 PHT_State[4,6]:=0;
   		 PHT_State[5,0]:=0;
   		 PHT_State[5,1]:=0;
   		 PHT_State[5,2]:=0;
   		 PHT_State[5,3]:=0;
   		 PHT_State[5,4]:=0;
   		 PHT_State[5,5]:=0;
   		 PHT_State[5,6]:=0;
   		 PHT_State[6,0]:=0;
   		 PHT_State[6,1]:=3;
   		 PHT_State[6,2]:=0;
   		 PHT_State[6,3]:=0;
   		 PHT_State[6,4]:=4;
   		 PHT_State[6,5]:=0;
   		 PHT_State[6,6]:=4;
   		 PHT_Table[0,0,0]:=207173177;
   		 PHT_Table[1,0,0]:=95901857;
   		 PHT_Table[2,0,0]:=243847721;
   		 PHT_Table[3,0,0]:=212974363;
   		 PHT_Table[4,0,0]:=210906504;
   		 PHT_Table[5,0,0]:=236619131;
   		 PHT_Table[6,0,0]:=9354536;
   		 PHT_Table[0,1,0]:=91409346;
   		 PHT_Table[1,1,0]:=128939748;
   		 PHT_Table[2,1,0]:=224794754;
   		 PHT_Table[3,1,0]:=94677578;
   		 PHT_Table[4,1,0]:=86540646;
   		 PHT_Table[5,1,0]:=223242234;
   		 PHT_Table[6,1,0]:=12037226;
   		 PHT_Table[0,2,0]:=113083277;
   		 PHT_Table[1,2,0]:=197833817;
   		 PHT_Table[2,2,0]:=121958685;
   		 PHT_Table[3,2,0]:=113888412;
   		 PHT_Table[4,2,0]:=114368324;
   		 PHT_Table[5,2,0]:=127224748;
   		 PHT_Table[6,2,0]:=19871970;
   		 PHT_Table[0,3,0]:=195128417;
   		 PHT_Table[1,3,0]:=173974386;
   		 PHT_Table[2,3,0]:=255038529;
   		 PHT_Table[3,3,0]:=189945125;
   		 PHT_Table[4,3,0]:=185878835;
   		 PHT_Table[5,3,0]:=254229221;
   		 PHT_Table[6,3,0]:=16926466;
   		 PHT_Table[0,4,0]:=153878011;
   		 PHT_Table[1,4,0]:=35139141;
   		 PHT_Table[2,4,0]:=65981099;
   		 PHT_Table[3,4,0]:=152375633;
   		 PHT_Table[4,4,0]:=163228910;
   		 PHT_Table[5,4,0]:=55894657;
   		 PHT_Table[6,4,0]:=4612907;
   		 PHT_Table[0,5,0]:=0;
   		 PHT_Table[1,5,0]:=0;
   		 PHT_Table[2,5,0]:=0;
   		 PHT_Table[3,5,0]:=0;
   		 PHT_Table[4,5,0]:=0;
   		 PHT_Table[5,5,0]:=0;
   		 PHT_Table[6,5,0]:=0;
   		 PHT_Table[0,6,0]:=182760884;
   		 PHT_Table[1,6,0]:=243133688;
   		 PHT_Table[2,6,0]:=164373300;
   		 PHT_Table[3,6,0]:=175667079;
   		 PHT_Table[4,6,0]:=172176076;
   		 PHT_Table[5,6,0]:=160419543;
   		 PHT_Table[6,6,0]:=23981959;
   		 PHT_Table[0,7,0]:=220000236;
   		 PHT_Table[1,7,0]:=26482475;
   		 PHT_Table[2,7,0]:=142042460;
   		 PHT_Table[3,7,0]:=228301241;
   		 PHT_Table[4,7,0]:=231036535;
   		 PHT_Table[5,7,0]:=145912137;
   		 PHT_Table[6,7,0]:=3034284;
   		 PHT_Table[0,8,0]:=63916111;
   		 PHT_Table[1,8,0]:=207995581;
   		 PHT_Table[2,8,0]:=170060191;
   		 PHT_Table[3,8,0]:=57501398;
   		 PHT_Table[4,8,0]:=66690594;
   		 PHT_Table[5,8,0]:=182135894;
   		 PHT_Table[6,8,0]:=21735142;
   		 PHT_Table[0,9,0]:=248752035;
   		 PHT_Table[1,9,0]:=233952662;
   		 PHT_Table[2,9,0]:=39161027;
   		 PHT_Table[3,9,0]:=251068271;
   		 PHT_Table[4,9,0]:=238864469;
   		 PHT_Table[5,9,0]:=40459551;
   		 PHT_Table[6,9,0]:=22193618;
   		 PHT_Table[0,10,0]:=261521014;
   		 PHT_Table[1,10,0]:=164796956;
   		 PHT_Table[2,10,0]:=78265270;
   		 PHT_Table[3,10,0]:=266132941;
   		 PHT_Table[4,10,0]:=258716586;
   		 PHT_Table[5,10,0]:=79800621;
   		 PHT_Table[6,10,0]:=15780439;
   		 PHT_Table[0,11,0]:=141435950;
   		 PHT_Table[1,11,0]:=104554959;
   		 PHT_Table[2,11,0]:=85032414;
   		 PHT_Table[3,11,0]:=138359795;
   		 PHT_Table[4,11,0]:=149804817;
   		 PHT_Table[5,11,0]:=100406963;
   		 PHT_Table[6,11,0]:=11549155;
   		 PHT_Table[0,12,0]:=70717975;
   		 PHT_Table[1,12,0]:=59521390;
   		 PHT_Table[2,12,0]:=194621431;
   		 PHT_Table[3,12,0]:=76450024;
   		 PHT_Table[4,12,0]:=75496089;
   		 PHT_Table[5,12,0]:=199660488;
   		 PHT_Table[6,12,0]:=5774577;
   		 PHT_Table[0,13,0]:=133716568;
   		 PHT_Table[1,13,0]:=266992595;
   		 PHT_Table[2,13,0]:=29050472;
   		 PHT_Table[3,13,0]:=132378174;
   		 PHT_Table[4,13,0]:=126248123;
   		 PHT_Table[5,13,0]:=20823966;
   		 PHT_Table[6,13,0]:=26041691;
   		 PHT_Table[0,14,0]:=21354965;
   		 PHT_Table[1,14,0]:=69422986;
   		 PHT_Table[2,14,0]:=117421941;
   		 PHT_Table[3,14,0]:=19538594;
   		 PHT_Table[4,14,0]:=22510591;
   		 PHT_Table[5,14,0]:=111735858;
   		 PHT_Table[6,14,0]:=7324398;
   		 PHT_Table[0,15,0]:=42635674;
   		 PHT_Table[1,15,0]:=138841399;
   		 PHT_Table[2,15,0]:=215834346;
   		 PHT_Table[3,15,0]:=38225012;
   		 PHT_Table[4,15,0]:=45016541;
   		 PHT_Table[5,15,0]:=208918628;
   		 PHT_Table[6,15,0]:=14529988;
   	 4:
   		PHT_D:=8;
   		PHT_S:=4;
   		PHT_RATE:=32;
   		PHT_RATEP:=32;
   		PHT_DIGESTSIZE:=224;
   		 PHT_RC[0,0]:=1;
   		 PHT_RC[0,1]:=3;
   		 PHT_RC[0,2]:=7;
   		 PHT_RC[0,3]:=14;
   		 PHT_RC[0,4]:=13;
   		 PHT_RC[0,5]:=11;
   		 PHT_RC[0,6]:=6;
   		 PHT_RC[0,7]:=12;
   		 PHT_RC[0,8]:=9;
   		 PHT_RC[0,9]:=2;
   		 PHT_RC[0,10]:=5;
   		 PHT_RC[0,11]:=10;
   		 PHT_RC[1,0]:=0;
   		 PHT_RC[1,1]:=2;
   		 PHT_RC[1,2]:=6;
   		 PHT_RC[1,3]:=15;
   		 PHT_RC[1,4]:=12;
   		 PHT_RC[1,5]:=10;
   		 PHT_RC[1,6]:=7;
   		 PHT_RC[1,7]:=13;
   		 PHT_RC[1,8]:=8;
   		 PHT_RC[1,9]:=3;
   		 PHT_RC[1,10]:=4;
   		 PHT_RC[1,11]:=11;
   		 PHT_RC[2,0]:=2;
   		 PHT_RC[2,1]:=0;
   		 PHT_RC[2,2]:=4;
   		 PHT_RC[2,3]:=13;
   		 PHT_RC[2,4]:=14;
   		 PHT_RC[2,5]:=8;
   		 PHT_RC[2,6]:=5;
   		 PHT_RC[2,7]:=15;
   		 PHT_RC[2,8]:=10;
   		 PHT_RC[2,9]:=1;
   		 PHT_RC[2,10]:=6;
   		 PHT_RC[2,11]:=9;
   		 PHT_RC[3,0]:=6;
   		 PHT_RC[3,1]:=4;
   		 PHT_RC[3,2]:=0;
   		 PHT_RC[3,3]:=9;
   		 PHT_RC[3,4]:=10;
   		 PHT_RC[3,5]:=12;
   		 PHT_RC[3,6]:=1;
   		 PHT_RC[3,7]:=11;
   		 PHT_RC[3,8]:=14;
   		 PHT_RC[3,9]:=5;
   		 PHT_RC[3,10]:=2;
   		 PHT_RC[3,11]:=13;
   		 PHT_RC[4,0]:=14;
   		 PHT_RC[4,1]:=12;
   		 PHT_RC[4,2]:=8;
   		 PHT_RC[4,3]:=1;
   		 PHT_RC[4,4]:=2;
   		 PHT_RC[4,5]:=4;
   		 PHT_RC[4,6]:=9;
   		 PHT_RC[4,7]:=3;
   		 PHT_RC[4,8]:=6;
   		 PHT_RC[4,9]:=13;
   		 PHT_RC[4,10]:=10;
   		 PHT_RC[4,11]:=5;
   		 PHT_RC[5,0]:=15;
   		 PHT_RC[5,1]:=13;
   		 PHT_RC[5,2]:=9;
   		 PHT_RC[5,3]:=0;
   		 PHT_RC[5,4]:=3;
   		 PHT_RC[5,5]:=5;
   		 PHT_RC[5,6]:=8;
   		 PHT_RC[5,7]:=2;
   		 PHT_RC[5,8]:=7;
   		 PHT_RC[5,9]:=12;
   		 PHT_RC[5,10]:=11;
   		 PHT_RC[5,11]:=4;
   		 PHT_RC[6,0]:=13;
   		 PHT_RC[6,1]:=15;
   		 PHT_RC[6,2]:=11;
   		 PHT_RC[6,3]:=2;
   		 PHT_RC[6,4]:=1;
   		 PHT_RC[6,5]:=7;
   		 PHT_RC[6,6]:=10;
   		 PHT_RC[6,7]:=0;
   		 PHT_RC[6,8]:=5;
   		 PHT_RC[6,9]:=14;
   		 PHT_RC[6,10]:=9;
   		 PHT_RC[6,11]:=6;
   		 PHT_RC[7,0]:=9;
   		 PHT_RC[7,1]:=11;
   		 PHT_RC[7,2]:=15;
   		 PHT_RC[7,3]:=6;
   		 PHT_RC[7,4]:=5;
   		 PHT_RC[7,5]:=3;
   		 PHT_RC[7,6]:=14;
   		 PHT_RC[7,7]:=4;
   		 PHT_RC[7,8]:=1;
   		 PHT_RC[7,9]:=10;
   		 PHT_RC[7,10]:=13;
   		 PHT_RC[7,11]:=2;
   		 PHT_State[0,0]:=0;
   		 PHT_State[0,1]:=0;
   		 PHT_State[0,2]:=0;
   		 PHT_State[0,3]:=0;
   		 PHT_State[0,4]:=0;
   		 PHT_State[0,5]:=0;
   		 PHT_State[0,6]:=0;
   		 PHT_State[0,7]:=0;
   		 PHT_State[1,0]:=0;
   		 PHT_State[1,1]:=0;
   		 PHT_State[1,2]:=0;
   		 PHT_State[1,3]:=0;
   		 PHT_State[1,4]:=0;
   		 PHT_State[1,5]:=0;
   		 PHT_State[1,6]:=0;
   		 PHT_State[1,7]:=0;
   		 PHT_State[2,0]:=0;
   		 PHT_State[2,1]:=0;
   		 PHT_State[2,2]:=0;
   		 PHT_State[2,3]:=0;
   		 PHT_State[2,4]:=0;
   		 PHT_State[2,5]:=0;
   		 PHT_State[2,6]:=0;
   		 PHT_State[2,7]:=0;
   		 PHT_State[3,0]:=0;
   		 PHT_State[3,1]:=0;
   		 PHT_State[3,2]:=0;
   		 PHT_State[3,3]:=0;
   		 PHT_State[3,4]:=0;
   		 PHT_State[3,5]:=0;
   		 PHT_State[3,6]:=0;
   		 PHT_State[3,7]:=0;
   		 PHT_State[4,0]:=0;
   		 PHT_State[4,1]:=0;
   		 PHT_State[4,2]:=0;
   		 PHT_State[4,3]:=0;
   		 PHT_State[4,4]:=0;
   		 PHT_State[4,5]:=0;
   		 PHT_State[4,6]:=0;
   		 PHT_State[4,7]:=0;
   		 PHT_State[5,0]:=0;
   		 PHT_State[5,1]:=0;
   		 PHT_State[5,2]:=0;
   		 PHT_State[5,3]:=0;
   		 PHT_State[5,4]:=0;
   		 PHT_State[5,5]:=0;
   		 PHT_State[5,6]:=0;
   		 PHT_State[5,7]:=0;
   		 PHT_State[6,0]:=0;
   		 PHT_State[6,1]:=0;
   		 PHT_State[6,2]:=0;
   		 PHT_State[6,3]:=0;
   		 PHT_State[6,4]:=0;
   		 PHT_State[6,5]:=0;
   		 PHT_State[6,6]:=0;
   		 PHT_State[6,7]:=0;
   		 PHT_State[7,0]:=0;
   		 PHT_State[7,1]:=0;
   		 PHT_State[7,2]:=3;
   		 PHT_State[7,3]:=8;
   		 PHT_State[7,4]:=2;
   		 PHT_State[7,5]:=0;
   		 PHT_State[7,6]:=2;
   		 PHT_State[7,7]:=0;
   		 PHT_Table[0,0,0]:=-1084455176;
   		 PHT_Table[1,0,0]:=1449063612;
   		 PHT_Table[2,0,0]:=-1170642509;
   		 PHT_Table[3,0,0]:=-751028207;
   		 PHT_Table[4,0,0]:=-1301330567;
   		 PHT_Table[5,0,0]:=-1571577919;
   		 PHT_Table[6,0,0]:=-1724365109;
   		 PHT_Table[7,0,0]:=-345751993;
   		 PHT_Table[0,1,0]:=-1451922538;
   		 PHT_Table[1,1,0]:=2071827365;
   		 PHT_Table[2,1,0]:=-1362971988;
   		 PHT_Table[3,1,0]:=482723396;
   		 PHT_Table[4,1,0]:=-1464256526;
   		 PHT_Table[5,1,0]:=-394516140;
   		 PHT_Table[6,1,0]:=583416666;
   		 PHT_Table[7,1,0]:=-625750721;
   		 PHT_Table[0,2,0]:=-826915868;
   		 PHT_Table[1,2,0]:=-1279794490;
   		 PHT_Table[2,2,0]:=-980599352;
   		 PHT_Table[3,2,0]:=-125401959;
   		 PHT_Table[4,2,0]:=-1052890195;
   		 PHT_Table[5,2,0]:=1371070057;
   		 PHT_Table[6,2,0]:=-578542740;
   		 PHT_Table[7,2,0]:=2083686186;
   		 PHT_Table[0,3,0]:=1571503315;
   		 PHT_Table[1,3,0]:=-1397761957;
   		 PHT_Table[2,3,0]:=1466024278;
   		 PHT_Table[3,3,0]:=-1771347166;
   		 PHT_Table[4,3,0]:=1422756577;
   		 PHT_Table[5,3,0]:=1957043634;
   		 PHT_Table[6,3,0]:=291736757;
   		 PHT_Table[7,3,0]:=-171413618;
   		 PHT_Table[0,4,0]:=371846510;
   		 PHT_Table[1,4,0]:=757294873;
   		 PHT_Table[2,4,0]:=352049951;
   		 PHT_Table[3,4,0]:=-805700011;
   		 PHT_Table[4,4,0]:=450261643;
   		 PHT_Table[5,4,0]:=1244640917;
   		 PHT_Table[6,4,0]:=-1140949615;
   		 PHT_Table[7,4,0]:=836236152;
   		 PHT_Table[0,5,0]:=0;
   		 PHT_Table[1,5,0]:=0;
   		 PHT_Table[2,5,0]:=0;
   		 PHT_Table[3,5,0]:=0;
   		 PHT_Table[4,5,0]:=0;
   		 PHT_Table[5,5,0]:=0;
   		 PHT_Table[6,5,0]:=0;
   		 PHT_Table[7,5,0]:=0;
   		 PHT_Table[0,6,0]:=1911211292;
   		 PHT_Table[1,6,0]:=-437709190;
   		 PHT_Table[2,6,0]:=2142524539;
   		 PHT_Table[3,6,0]:=733658248;
   		 PHT_Table[4,6,0]:=1934716628;
   		 PHT_Table[5,6,0]:=-202686040;
   		 PHT_Table[6,6,0]:=1153197479;
   		 PHT_Table[7,6,0]:=-1755924115;
   		 PHT_Table[0,7,0]:=-1826783433;
   		 PHT_Table[1,7,0]:=521681565;
   		 PHT_Table[2,7,0]:=-1829962594;
   		 PHT_Table[3,7,0]:=1861085115;
   		 PHT_Table[4,7,0]:=-1779195572;
   		 PHT_Table[5,7,0]:=622773211;
   		 PHT_Table[6,7,0]:=-857231399;
   		 PHT_Table[7,7,0]:=-1980045148;
   		 PHT_Table[0,8,0]:=1740843122;
   		 PHT_Table[1,8,0]:=-926256797;
   		 PHT_Table[2,8,0]:=1800376164;
   		 PHT_Table[3,8,0]:=-465354019;
   		 PHT_Table[4,8,0]:=1770462303;
   		 PHT_Table[5,8,0]:=-1178273987;
   		 PHT_Table[6,8,0]:=-12445642;
   		 PHT_Table[7,8,0]:=-1501476331;
   		 PHT_Table[0,9,0]:=-186755259;
   		 PHT_Table[1,9,0]:=-674083842;
   		 PHT_Table[2,9,0]:=-106728454;
   		 PHT_Table[3,9,0]:=-1968265882;
   		 PHT_Table[4,9,0]:=-59458285;
   		 PHT_Table[5,9,0]:=-1663421210;
   		 PHT_Table[6,9,0]:=866498543;
   		 PHT_Table[7,9,0]:=796631729;
   		 PHT_Table[0,10,0]:=-660623734;
   		 PHT_Table[1,10,0]:=-1634433569;
   		 PHT_Table[2,10,0]:=-780736809;
   		 PHT_Table[3,10,0]:=931101388;
   		 PHT_Table[4,10,0]:=-605529818;
   		 PHT_Table[5,10,0]:=462907644;
   		 PHT_Table[6,10,0]:=1719295741;
   		 PHT_Table[7,10,0]:=1306883154;
   		 PHT_Table[0,11,0]:=979899553;
   		 PHT_Table[1,11,0]:=1684384056;
   		 PHT_Table[2,11,0]:=1009667634;
   		 PHT_Table[3,11,0]:=1915232767;
   		 PHT_Table[4,11,0]:=1028298430;
   		 PHT_Table[5,11,0]:=-849155441;
   		 PHT_Table[6,11,0]:=-299789181;
   		 PHT_Table[7,11,0]:=1397302683;
   		 PHT_Table[0,12,0]:=-2060152231;
   		 PHT_Table[1,12,0]:=842751364;
   		 PHT_Table[2,12,0]:=-2045302911;
   		 PHT_Table[3,12,0]:=-1592518162;
   		 PHT_Table[4,12,0]:=-1893346361;
   		 PHT_Table[5,12,0]:=1865512270;
   		 PHT_Table[6,12,0]:=1998180936;
   		 PHT_Table[7,12,0]:=-1205003300;
   		 PHT_Table[0,13,0]:=-487081429;
   		 PHT_Table[1,13,0]:=-84857625;
   		 PHT_Table[2,13,0]:=-312956699;
   		 PHT_Table[3,13,0]:=1163352883;
   		 PHT_Table[4,13,0]:=-425537640;
   		 PHT_Table[5,13,0]:=-688553357;
   		 PHT_Table[6,13,0]:=-2007250306;
   		 PHT_Table[7,13,0]:=514609609;
   		 PHT_Table[0,14,0]:=742521295;
   		 PHT_Table[1,14,0]:=1229377057;
   		 PHT_Table[2,14,0]:=685085997;
   		 PHT_Table[3,14,0]:=-1110319190;
   		 PHT_Table[4,14,0]:=664593461;
   		 PHT_Table[5,14,0]:=-2024973286;
   		 PHT_Table[6,14,0]:=1440737554;
   		 PHT_Table[7,14,0]:=1654576867;
   		 PHT_Table[0,15,0]:=1266864573;
   		 PHT_Table[1,15,0]:=-2121482430;
   		 PHT_Table[2,15,0]:=1134172745;
   		 PHT_Table[3,15,0]:=1502780791;
   		 PHT_Table[4,15,0]:=1310455914;
   		 PHT_Table[5,15,0]:=1049209639;
   		 PHT_Table[6,15,0]:=-1432489692;
   		 PHT_Table[7,15,0]:=-1004561162;
   	 5:
   		PHT_D:=6;
   		PHT_S:=8;
   		PHT_RATE:=32;
   		PHT_RATEP:=32;
   		PHT_DIGESTSIZE:=256;
   		 PHT_RC[0,0]:=1;
   		 PHT_RC[0,1]:=3;
   		 PHT_RC[0,2]:=7;
   		 PHT_RC[0,3]:=14;
   		 PHT_RC[0,4]:=13;
   		 PHT_RC[0,5]:=11;
   		 PHT_RC[0,6]:=6;
   		 PHT_RC[0,7]:=12;
   		 PHT_RC[0,8]:=9;
   		 PHT_RC[0,9]:=2;
   		 PHT_RC[0,10]:=5;
   		 PHT_RC[0,11]:=10;
   		 PHT_RC[1,0]:=0;
   		 PHT_RC[1,1]:=2;
   		 PHT_RC[1,2]:=6;
   		 PHT_RC[1,3]:=15;
   		 PHT_RC[1,4]:=12;
   		 PHT_RC[1,5]:=10;
   		 PHT_RC[1,6]:=7;
   		 PHT_RC[1,7]:=13;
   		 PHT_RC[1,8]:=8;
   		 PHT_RC[1,9]:=3;
   		 PHT_RC[1,10]:=4;
   		 PHT_RC[1,11]:=11;
   		 PHT_RC[2,0]:=2;
   		 PHT_RC[2,1]:=0;
   		 PHT_RC[2,2]:=4;
   		 PHT_RC[2,3]:=13;
   		 PHT_RC[2,4]:=14;
   		 PHT_RC[2,5]:=8;
   		 PHT_RC[2,6]:=5;
   		 PHT_RC[2,7]:=15;
   		 PHT_RC[2,8]:=10;
   		 PHT_RC[2,9]:=1;
   		 PHT_RC[2,10]:=6;
   		 PHT_RC[2,11]:=9;
   		 PHT_RC[3,0]:=6;
   		 PHT_RC[3,1]:=4;
   		 PHT_RC[3,2]:=0;
   		 PHT_RC[3,3]:=9;
   		 PHT_RC[3,4]:=10;
   		 PHT_RC[3,5]:=12;
   		 PHT_RC[3,6]:=1;
   		 PHT_RC[3,7]:=11;
   		 PHT_RC[3,8]:=14;
   		 PHT_RC[3,9]:=5;
   		 PHT_RC[3,10]:=2;
   		 PHT_RC[3,11]:=13;
   		 PHT_RC[4,0]:=7;
   		 PHT_RC[4,1]:=5;
   		 PHT_RC[4,2]:=1;
   		 PHT_RC[4,3]:=8;
   		 PHT_RC[4,4]:=11;
   		 PHT_RC[4,5]:=13;
   		 PHT_RC[4,6]:=0;
   		 PHT_RC[4,7]:=10;
   		 PHT_RC[4,8]:=15;
   		 PHT_RC[4,9]:=4;
   		 PHT_RC[4,10]:=3;
   		 PHT_RC[4,11]:=12;
   		 PHT_RC[5,0]:=5;
   		 PHT_RC[5,1]:=7;
   		 PHT_RC[5,2]:=3;
   		 PHT_RC[5,3]:=10;
   		 PHT_RC[5,4]:=9;
   		 PHT_RC[5,5]:=15;
   		 PHT_RC[5,6]:=2;
   		 PHT_RC[5,7]:=8;
   		 PHT_RC[5,8]:=13;
   		 PHT_RC[5,9]:=6;
   		 PHT_RC[5,10]:=1;
   		 PHT_RC[5,11]:=14;
   		 PHT_State[0,0]:=0;
   		 PHT_State[0,1]:=0;
   		 PHT_State[0,2]:=0;
   		 PHT_State[0,3]:=0;
   		 PHT_State[0,4]:=0;
   		 PHT_State[0,5]:=0;
   		 PHT_State[1,0]:=0;
   		 PHT_State[1,1]:=0;
   		 PHT_State[1,2]:=0;
   		 PHT_State[1,3]:=0;
   		 PHT_State[1,4]:=0;
   		 PHT_State[1,5]:=0;
   		 PHT_State[2,0]:=0;
   		 PHT_State[2,1]:=0;
   		 PHT_State[2,2]:=0;
   		 PHT_State[2,3]:=0;
   		 PHT_State[2,4]:=0;
   		 PHT_State[2,5]:=0;
   		 PHT_State[3,0]:=0;
   		 PHT_State[3,1]:=0;
   		 PHT_State[3,2]:=0;
   		 PHT_State[3,3]:=0;
   		 PHT_State[3,4]:=0;
   		 PHT_State[3,5]:=0;
   		 PHT_State[4,0]:=0;
   		 PHT_State[4,1]:=0;
   		 PHT_State[4,2]:=0;
   		 PHT_State[4,3]:=0;
   		 PHT_State[4,4]:=0;
   		 PHT_State[4,5]:=0;
   		 PHT_State[5,0]:=0;
   		 PHT_State[5,1]:=0;
   		 PHT_State[5,2]:=0;
   		 PHT_State[5,3]:=64;
   		 PHT_State[5,4]:=32;
   		 PHT_State[5,5]:=32;
   		 PHT_Table[0,0,0]:=317340486;
   		 PHT_Table[0,0,1]:=50741;
   		 PHT_Table[1,0,0]:=781009246;
   		 PHT_Table[1,0,1]:=42340;
   		 PHT_Table[2,0,0]:=1834687842;
   		 PHT_Table[2,0,1]:=25394;
   		 PHT_Table[3,0,0]:=545742939;
   		 PHT_Table[3,0,1]:=50774;
   		 PHT_Table[4,0,0]:=1599412035;
   		 PHT_Table[4,0,1]:=25425;
   		 PHT_Table[5,0,0]:=1972380571;
   		 PHT_Table[5,0,1]:=38665;
   		 PHT_Table[0,1,0]:=-510684426;
   		 PHT_Table[0,1,1]:=63693;
   		 PHT_Table[1,1,0]:=-777759713;
   		 PHT_Table[1,1,1]:=34014;
   		 PHT_Table[2,1,0]:=589032751;
   		 PHT_Table[2,1,1]:=31855;
   		 PHT_Table[3,1,0]:=-1901295333;
   		 PHT_Table[3,1,1]:=63665;
   		 PHT_Table[4,1,0]:=1279583730;
   		 PHT_Table[4,1,1]:=31763;
   		 PHT_Table[5,1,0]:=-901154030;
   		 PHT_Table[5,1,1]:=60413;
   		 PHT_Table[0,2,0]:=-1940645749;
   		 PHT_Table[0,2,1]:=61077;
   		 PHT_Table[1,2,0]:=1609711707;
   		 PHT_Table[1,2,1]:=39356;
   		 PHT_Table[2,2,0]:=-92930424;
   		 PHT_Table[2,2,1]:=30558;
   		 PHT_Table[3,2,0]:=-760320651;
   		 PHT_Table[3,2,1]:=61154;
   		 PHT_Table[4,2,0]:=-1527209307;
   		 PHT_Table[4,2,1]:=30505;
   		 PHT_Table[5,2,0]:=705480879;
   		 PHT_Table[5,2,1]:=51014;
   		 PHT_Table[0,3,0]:=255782969;
   		 PHT_Table[0,3,1]:=63221;
   		 PHT_Table[1,3,0]:=1882109528;
   		 PHT_Table[1,3,1]:=36340;
   		 PHT_Table[2,3,0]:=2121225767;
   		 PHT_Table[2,3,1]:=31610;
   		 PHT_Table[3,3,0]:=1967169391;
   		 PHT_Table[3,3,1]:=63118;
   		 PHT_Table[4,3,0]:=74070030;
   		 PHT_Table[4,3,1]:=31489;
   		 PHT_Table[5,3,0]:=527995210;
   		 PHT_Table[5,3,1]:=63370;
   		 PHT_Table[0,4,0]:=-1772444900;
   		 PHT_Table[0,4,1]:=65489;
   		 PHT_Table[1,4,0]:=216081841;
   		 PHT_Table[1,4,1]:=3531;
   		 PHT_Table[2,4,0]:=-2145305301;
   		 PHT_Table[2,4,1]:=62184;
   		 PHT_Table[3,4,0]:=2128249377;
   		 PHT_Table[3,4,1]:=65315;
   		 PHT_Table[4,4,0]:=1750271628;
   		 PHT_Table[4,4,1]:=61978;
   		 PHT_Table[5,4,0]:=769396286;
   		 PHT_Table[5,4,1]:=58699;
   		 PHT_Table[0,5,0]:=430345114;
   		 PHT_Table[0,5,1]:=54901;
   		 PHT_Table[1,5,0]:=-303241892;
   		 PHT_Table[1,5,1]:=48404;
   		 PHT_Table[2,5,0]:=-1782700888;
   		 PHT_Table[2,5,1]:=27402;
   		 PHT_Table[3,5,0]:=322123198;
   		 PHT_Table[3,5,1]:=54814;
   		 PHT_Table[4,5,0]:=-1623131272;
   		 PHT_Table[4,5,1]:=27489;
   		 PHT_Table[5,5,0]:=1405636052;
   		 PHT_Table[5,5,1]:=46977;
   		 PHT_Table[0,6,0]:=-1853828108;
   		 PHT_Table[0,6,1]:=56917;
   		 PHT_Table[1,6,0]:=22132573;
   		 PHT_Table[1,6,1]:=45356;
   		 PHT_Table[2,6,0]:=-381569587;
   		 PHT_Table[2,6,1]:=28438;
   		 PHT_Table[3,6,0]:=-2023124415;
   		 PHT_Table[3,6,1]:=56890;
   		 PHT_Table[4,6,0]:=-3699224;
   		 PHT_Table[4,6,1]:=28537;
   		 PHT_Table[5,6,0]:=1088715390;
   		 PHT_Table[5,6,1]:=42949;
   		 PHT_Table[0,7,0]:=1113082925;
   		 PHT_Table[0,7,1]:=37234;
   		 PHT_Table[1,7,0]:=288764666;
   		 PHT_Table[1,7,1]:=21722;
   		 PHT_Table[2,7,0]:=-79884119;
   		 PHT_Table[2,7,1]:=50541;
   		 PHT_Table[3,7,0]:=799240509;
   		 PHT_Table[3,7,1]:=37303;
   		 PHT_Table[4,7,0]:=-1778154006;
   		 PHT_Table[4,7,1]:=50600;
   		 PHT_Table[5,7,0]:=740727775;
   		 PHT_Table[5,7,1]:=14625;
   		 PHT_Table[0,8,0]:=984845822;
   		 PHT_Table[0,8,1]:=24731;
   		 PHT_Table[1,8,0]:=-1134693108;
   		 PHT_Table[1,8,1]:=20539;
   		 PHT_Table[2,8,0]:=644388490;
   		 PHT_Table[2,8,1]:=12432;
   		 PHT_Table[3,8,0]:=-1433016984;
   		 PHT_Table[3,8,1]:=24747;
   		 PHT_Table[4,8,0]:=-1233232230;
   		 PHT_Table[4,8,1]:=12448;
   		 PHT_Table[5,8,0]:=-724860999;
   		 PHT_Table[5,8,1]:=49181;
   		 PHT_Table[0,9,0]:=579081878;
   		 PHT_Table[0,9,1]:=520;
   		 PHT_Table[1,9,0]:=1004837323;
   		 PHT_Table[1,9,1]:=782;
   		 PHT_Table[2,9,0]:=528084946;
   		 PHT_Table[2,9,1]:=263;
   		 PHT_Table[3,9,0]:=630943609;
   		 PHT_Table[3,9,1]:=521;
   		 PHT_Table[4,9,0]:=409440292;
   		 PHT_Table[4,9,1]:=262;
   		 PHT_Table[5,9,0]:=1108036519;
   		 PHT_Table[5,9,1]:=1041;
   		 PHT_Table[0,10,0]:=-1697881304;
   		 PHT_Table[0,10,1]:=52757;
   		 PHT_Table[1,10,0]:=-1037036705;
   		 PHT_Table[1,10,1]:=43356;
   		 PHT_Table[2,10,0]:=295996423;
   		 PHT_Table[2,10,1]:=26414;
   		 PHT_Table[3,10,0]:=-1260533852;
   		 PHT_Table[3,10,1]:=52850;
   		 PHT_Table[4,10,0]:=1070752211;
   		 PHT_Table[4,10,1]:=26441;
   		 PHT_Table[5,10,0]:=1723601969;
   		 PHT_Table[5,10,1]:=34637;
   		 PHT_Table[0,11,0]:=1106279456;
   		 PHT_Table[0,11,1]:=22083;
   		 PHT_Table[1,11,0]:=-1345736116;
   		 PHT_Table[1,11,1]:=32185;
   		 PHT_Table[2,11,0]:=349697954;
   		 PHT_Table[2,11,1]:=11217;
   		 PHT_Table[3,11,0]:=-1864061993;
   		 PHT_Table[3,11,1]:=22120;
   		 PHT_Table[4,11,0]:=-974595397;
   		 PHT_Table[4,11,1]:=11258;
   		 PHT_Table[5,11,0]:=2017333402;
   		 PHT_Table[5,11,1]:=44205;
   		 PHT_Table[0,12,0]:=355486638;
   		 PHT_Table[0,12,1]:=59313;
   		 PHT_Table[1,12,0]:=591254450;
   		 PHT_Table[1,12,1]:=6531;
   		 PHT_Table[2,12,0]:=71013764;
   		 PHT_Table[2,12,1]:=65228;
   		 PHT_Table[3,12,0]:=-650874821;
   		 PHT_Table[3,12,1]:=59215;
   		 PHT_Table[4,12,0]:=-926835673;
   		 PHT_Table[4,12,1]:=65074;
   		 PHT_Table[5,12,0]:=413685723;
   		 PHT_Table[5,12,1]:=54663;
   		 PHT_Table[0,13,0]:=282270649;
   		 PHT_Table[0,13,1]:=46562;
   		 PHT_Table[1,13,0]:=-98088845;
   		 PHT_Table[1,13,1]:=25126;
   		 PHT_Table[2,13,0]:=773760921;
   		 PHT_Table[2,13,1]:=55059;
   		 PHT_Table[3,13,0]:=66913566;
   		 PHT_Table[3,13,1]:=46389;
   		 PHT_Table[4,13,0]:=1038581204;
   		 PHT_Table[4,13,1]:=55236;
   		 PHT_Table[5,13,0]:=-461319916;
   		 PHT_Table[5,13,1]:=28936;
   		 PHT_Table[0,14,0]:=-245593777;
   		 PHT_Table[0,14,1]:=19759;
   		 PHT_Table[1,14,0]:=730012780;
   		 PHT_Table[1,14,1]:=59128;
   		 PHT_Table[2,14,0]:=218450614;
   		 PHT_Table[2,14,1]:=43900;
   		 PHT_Table[3,14,0]:=-1924035579;
   		 PHT_Table[3,14,1]:=19844;
   		 PHT_Table[4,14,0]:=1906546726;
   		 PHT_Table[4,14,1]:=43991;
   		 PHT_Table[5,14,0]:=784968198;
   		 PHT_Table[5,14,1]:=39669;
   		 PHT_Table[0,15,0]:=-1362096611;
   		 PHT_Table[0,15,1]:=60573;
   		 PHT_Table[1,15,0]:=1679219088;
   		 PHT_Table[1,15,1]:=39602;
   		 PHT_Table[2,15,0]:=-452193958;
   		 PHT_Table[2,15,1]:=30297;
   		 PHT_Table[3,15,0]:=-147521012;
   		 PHT_Table[3,15,1]:=60651;
   		 PHT_Table[4,15,0]:=-1130417535;
   		 PHT_Table[4,15,1]:=30255;
   		 PHT_Table[5,15,0]:=1745322760;
   		 PHT_Table[5,15,1]:=50007;
   		 PHT_Table[0,16,0]:=-1482318274;
   		 PHT_Table[0,16,1]:=36618;
   		 PHT_Table[1,16,0]:=1943893183;
   		 PHT_Table[1,16,1]:=17792;
   		 PHT_Table[2,16,0]:=1588367979;
   		 PHT_Table[2,16,1]:=51776;
   		 PHT_Table[3,16,0]:=-402967892;
   		 PHT_Table[3,16,1]:=36800;
   		 PHT_Table[4,16,0]:=507032621;
   		 PHT_Table[4,16,1]:=51850;
   		 PHT_Table[5,16,0]:=-548462648;
   		 PHT_Table[5,16,1]:=1502;
   		 PHT_Table[0,17,0]:=-188753576;
   		 PHT_Table[0,17,1]:=8060;
   		 PHT_Table[1,17,0]:=-224819283;
   		 PHT_Table[1,17,1]:=40285;
   		 PHT_Table[2,17,0]:=656439467;
   		 PHT_Table[2,17,1]:=33443;
   		 PHT_Table[3,17,0]:=1469643040;
   		 PHT_Table[3,17,1]:=8190;
   		 PHT_Table[4,17,0]:=-2071627307;
   		 PHT_Table[4,17,1]:=33313;
   		 PHT_Table[5,17,0]:=-756994871;
   		 PHT_Table[5,17,1]:=15994;
   		 PHT_Table[0,18,0]:=-1053645665;
   		 PHT_Table[0,18,1]:=35090;
   		 PHT_Table[1,18,0]:=1055573241;
   		 PHT_Table[1,18,1]:=16530;
   		 PHT_Table[2,18,0]:=2133309446;
   		 PHT_Table[2,18,1]:=51529;
   		 PHT_Table[3,18,0]:=-2008186073;
   		 PHT_Table[3,18,1]:=35291;
   		 PHT_Table[4,18,0]:=915480385;
   		 PHT_Table[4,18,1]:=51584;
   		 PHT_Table[5,18,0]:=424854074;
   		 PHT_Table[5,18,1]:=2541;
   		 PHT_Table[0,19,0]:=-1022655392;
   		 PHT_Table[0,19,1]:=64197;
   		 PHT_Table[1,19,0]:=-364851756;
   		 PHT_Table[1,19,1]:=34768;
   		 PHT_Table[2,19,0]:=1013056253;
   		 PHT_Table[2,19,1]:=32104;
   		 PHT_Table[3,19,0]:=-1422399902;
   		 PHT_Table[3,19,1]:=64184;
   		 PHT_Table[4,19,0]:=1411610070;
   		 PHT_Table[4,19,1]:=32021;
   		 PHT_Table[5,19,0]:=-2008928075;
   		 PHT_Table[5,19,1]:=61420;
   		 PHT_Table[0,20,0]:=-1659497536;
   		 PHT_Table[0,20,1]:=61329;
   		 PHT_Table[1,20,0]:=-813661773;
   		 PHT_Table[1,20,1]:=5563;
   		 PHT_Table[2,20,0]:=2026112225;
   		 PHT_Table[2,20,1]:=64208;
   		 PHT_Table[3,20,0]:=1299109828;
   		 PHT_Table[3,20,1]:=61291;
   		 PHT_Table[4,20,0]:=-1471747401;
   		 PHT_Table[4,20,1]:=64042;
   		 PHT_Table[5,20,0]:=193224817;
   		 PHT_Table[5,20,1]:=50627;
   		 PHT_Table[0,21,0]:=1728457299;
   		 PHT_Table[0,21,1]:=45822;
   		 PHT_Table[1,21,0]:=660748765;
   		 PHT_Table[1,21,1]:=60211;
   		 PHT_Table[2,21,0]:=-1926989923;
   		 PHT_Table[2,21,1]:=22932;
   		 PHT_Table[3,21,0]:=-208990684;
   		 PHT_Table[3,21,1]:=45735;
   		 PHT_Table[4,21,0]:=435199658;
   		 PHT_Table[4,21,1]:=22989;
   		 PHT_Table[5,21,0]:=51749944;
   		 PHT_Table[5,21,1]:=32702;
   		 PHT_Table[0,22,0]:=-1226336907;
   		 PHT_Table[0,22,1]:=36366;
   		 PHT_Table[1,22,0]:=-475024041;
   		 PHT_Table[1,22,1]:=51591;
   		 PHT_Table[2,22,0]:=-602052606;
   		 PHT_Table[2,22,1]:=18382;
   		 PHT_Table[3,22,0]:=2017167389;
   		 PHT_Table[3,22,1]:=36425;
   		 PHT_Table[4,22,0]:=310836287;
   		 PHT_Table[4,22,1]:=18313;
   		 PHT_Table[5,22,0]:=-20465898;
   		 PHT_Table[5,22,1]:=1883;
   		 PHT_Table[0,23,0]:=-766931157;
   		 PHT_Table[0,23,1]:=64449;
   		 PHT_Table[1,23,0]:=2050100284;
   		 PHT_Table[1,23,1]:=3031;
   		 PHT_Table[2,23,0]:=-1093404524;
   		 PHT_Table[2,23,1]:=61670;
   		 PHT_Table[3,23,0]:=888626387;
   		 PHT_Table[3,23,1]:=64305;
   		 PHT_Table[4,23,0]:=1486699972;
   		 PHT_Table[4,23,1]:=61462;
   		 PHT_Table[5,23,0]:=-1446340501;
   		 PHT_Table[5,23,1]:=60777;
   		 PHT_Table[0,24,0]:=1030356246;
   		 PHT_Table[0,24,1]:=16671;
   		 PHT_Table[1,24,0]:=-1309841440;
   		 PHT_Table[1,24,1]:=60636;
   		 PHT_Table[2,24,0]:=1325932140;
   		 PHT_Table[2,24,1]:=44398;
   		 PHT_Table[3,24,0]:=1395062024;
   		 PHT_Table[3,24,1]:=16818;
   		 PHT_Table[4,24,0]:=569038334;
   		 PHT_Table[4,24,1]:=44483;
   		 PHT_Table[5,24,0]:=-1175254023;
   		 PHT_Table[5,24,1]:=33427;
   		 PHT_Table[0,25,0]:=1984176408;
   		 PHT_Table[0,25,1]:=46074;
   		 PHT_Table[1,25,0]:=-1223624651;
   		 PHT_Table[1,25,1]:=26420;
   		 PHT_Table[2,25,0]:=261459444;
   		 PHT_Table[2,25,1]:=54298;
   		 PHT_Table[3,25,0]:=1816900757;
   		 PHT_Table[3,25,1]:=45870;
   		 PHT_Table[4,25,0]:=357488312;
   		 PHT_Table[4,25,1]:=54478;
   		 PHT_Table[5,25,0]:=580717798;
   		 PHT_Table[5,25,1]:=32059;
   		 PHT_Table[0,26,0]:=-661377275;
   		 PHT_Table[0,26,1]:=24423;
   		 PHT_Table[1,26,0]:=-754572891;
   		 PHT_Table[1,26,1]:=64902;
   		 PHT_Table[2,26,0]:=-359031634;
   		 PHT_Table[2,26,1]:=41539;
   		 PHT_Table[3,26,0]:=-1686194535;
   		 PHT_Table[3,26,1]:=24517;
   		 PHT_Table[4,26,0]:=-1445862343;
   		 PHT_Table[4,26,1]:=41697;
   		 PHT_Table[5,26,0]:=1251643374;
   		 PHT_Table[5,26,1]:=48748;
   		 PHT_Table[0,27,0]:=2038092065;
   		 PHT_Table[0,27,1]:=17679;
   		 PHT_Table[1,27,0]:=-952218003;
   		 PHT_Table[1,27,1]:=60096;
   		 PHT_Table[2,27,0]:=1912265683;
   		 PHT_Table[2,27,1]:=44896;
   		 PHT_Table[3,27,0]:=420162554;
   		 PHT_Table[3,27,1]:=17824;
   		 PHT_Table[4,27,0]:=287633078;
   		 PHT_Table[4,27,1]:=45007;
   		 PHT_Table[5,27,0]:=1038458284;
   		 PHT_Table[5,27,1]:=35505;
   		 PHT_Table[0,28,0]:=626943614;
   		 PHT_Table[0,28,1]:=9100;
   		 PHT_Table[1,28,0]:=911477543;
   		 PHT_Table[1,28,1]:=49129;
   		 PHT_Table[2,28,0]:=1981376308;
   		 PHT_Table[2,28,1]:=40185;
   		 PHT_Table[3,28,0]:=-601325799;
   		 PHT_Table[3,28,1]:=8976;
   		 PHT_Table[4,28,0]:=-1879893184;
   		 PHT_Table[4,28,1]:=40037;
   		 PHT_Table[5,28,0]:=791887847;
   		 PHT_Table[5,28,1]:=18079;
   		 PHT_Table[0,29,0]:=346119004;
   		 PHT_Table[0,29,1]:=21335;
   		 PHT_Table[1,29,0]:=1231575593;
   		 PHT_Table[1,29,1]:=63394;
   		 PHT_Table[2,29,0]:=-1466644364;
   		 PHT_Table[2,29,1]:=42065;
   		 PHT_Table[3,29,0]:=1158270868;
   		 PHT_Table[3,29,1]:=21491;
   		 PHT_Table[4,29,0]:=-107435551;
   		 PHT_Table[4,29,1]:=42229;
   		 PHT_Table[5,29,0]:=-576705007;
   		 PHT_Table[5,29,1]:=42506;
   		 PHT_Table[0,30,0]:=653678195;
   		 PHT_Table[0,30,1]:=58557;
   		 PHT_Table[1,30,0]:=-2002023535;
   		 PHT_Table[1,30,1]:=38538;
   		 PHT_Table[2,30,0]:=-1712095169;
   		 PHT_Table[2,30,1]:=29253;
   		 PHT_Table[3,30,0]:=1668261363;
   		 PHT_Table[3,30,1]:=58575;
   		 PHT_Table[4,30,0]:=-602389487;
   		 PHT_Table[4,30,1]:=29239;
   		 PHT_Table[5,30,0]:=2066461858;
   		 PHT_Table[5,30,1]:=54035;
   		 PHT_Table[0,31,0]:=-386268459;
   		 PHT_Table[0,31,1]:=39770;
   		 PHT_Table[1,31,0]:=-965740240;
   		 PHT_Table[1,31,1]:=23532;
   		 PHT_Table[2,31,0]:=-1732547042;
   		 PHT_Table[2,31,1]:=49270;
   		 PHT_Table[3,31,0]:=-1637697093;
   		 PHT_Table[3,31,1]:=39834;
   		 PHT_Table[4,31,0]:=-287087778;
   		 PHT_Table[4,31,1]:=49334;
   		 PHT_Table[5,31,0]:=2097276882;
   		 PHT_Table[5,31,1]:=11636;
   		 PHT_Table[0,32,0]:=1689131614;
   		 PHT_Table[0,32,1]:=30159;
   		 PHT_Table[1,32,0]:=-1717716629;
   		 PHT_Table[1,32,1]:=49744;
   		 PHT_Table[2,32,0]:=1657704598;
   		 PHT_Table[2,32,1]:=46888;
   		 PHT_Table[3,32,0]:=1288492238;
   		 PHT_Table[3,32,1]:=30072;
   		 PHT_Table[4,32,0]:=1243333115;
   		 PHT_Table[4,32,1]:=47007;
   		 PHT_Table[5,32,0]:=1460481917;
   		 PHT_Table[5,32,1]:=59954;
   		 PHT_Table[0,33,0]:=1940353295;
   		 PHT_Table[0,33,1]:=57769;
   		 PHT_Table[1,33,0]:=1846174708;
   		 PHT_Table[1,33,1]:=7313;
   		 PHT_Table[2,33,0]:=632340457;
   		 PHT_Table[2,33,1]:=64965;
   		 PHT_Table[3,33,0]:=-1232944720;
   		 PHT_Table[3,33,1]:=57684;
   		 PHT_Table[4,33,0]:=-530041013;
   		 PHT_Table[4,33,1]:=64824;
   		 PHT_Table[5,33,0]:=-558527959;
   		 PHT_Table[5,33,1]:=55732;
   		 PHT_Table[0,34,0]:=-1063013267;
   		 PHT_Table[0,34,1]:=15860;
   		 PHT_Table[1,34,0]:=1421823330;
   		 PHT_Table[1,34,1]:=44723;
   		 PHT_Table[2,34,0]:=-746002954;
   		 PHT_Table[2,34,1]:=37844;
   		 PHT_Table[3,34,0]:=342899848;
   		 PHT_Table[3,34,1]:=15719;
   		 PHT_Table[4,34,0]:=130558599;
   		 PHT_Table[4,34,1]:=37703;
   		 PHT_Table[5,34,0]:=-598033424;
   		 PHT_Table[5,34,1]:=31328;
   		 PHT_Table[0,35,0]:=-534871548;
   		 PHT_Table[0,35,1]:=19499;
   		 PHT_Table[1,35,0]:=-1141777020;
   		 PHT_Table[1,35,1]:=27391;
   		 PHT_Table[2,35,0]:=-1883983649;
   		 PHT_Table[2,35,1]:=9970;
   		 PHT_Table[3,35,0]:=311506612;
   		 PHT_Table[3,35,1]:=19469;
   		 PHT_Table[4,35,0]:=2099105844;
   		 PHT_Table[4,35,1]:=9940;
   		 PHT_Table[5,35,0]:=255918808;
   		 PHT_Table[5,35,1]:=39024;
   		 PHT_Table[0,36,0]:=-158926425;
   		 PHT_Table[0,36,1]:=27819;
   		 PHT_Table[1,36,0]:=640913024;
   		 PHT_Table[1,36,1]:=23071;
   		 PHT_Table[2,36,0]:=1684390480;
   		 PHT_Table[2,36,1]:=13954;
   		 PHT_Table[3,36,0]:=1961008229;
   		 PHT_Table[3,36,1]:=27805;
   		 PHT_Table[4,36,0]:=-432598206;
   		 PHT_Table[4,36,1]:=14004;
   		 PHT_Table[5,36,0]:=1139924550;
   		 PHT_Table[5,36,1]:=55419;
   		 PHT_Table[0,37,0]:=-548511763;
   		 PHT_Table[0,37,1]:=32483;
   		 PHT_Table[1,37,0]:=-558451895;
   		 PHT_Table[1,37,1]:=16737;
   		 PHT_Table[2,37,0]:=-2080828344;
   		 PHT_Table[2,37,1]:=16317;
   		 PHT_Table[3,37,0]:=1657644793;
   		 PHT_Table[3,37,1]:=32476;
   		 PHT_Table[4,37,0]:=1044737885;
   		 PHT_Table[4,37,1]:=16258;
   		 PHT_Table[5,37,0]:=664992686;
   		 PHT_Table[5,37,1]:=64738;
   		 PHT_Table[0,38,0]:=1022946788;
   		 PHT_Table[0,38,1]:=62969;
   		 PHT_Table[1,38,0]:=-608637317;
   		 PHT_Table[1,38,1]:=765;
   		 PHT_Table[2,38,0]:=-475577444;
   		 PHT_Table[2,38,1]:=63475;
   		 PHT_Table[3,38,0]:=-820295001;
   		 PHT_Table[3,38,1]:=62734;
   		 PHT_Table[4,38,0]:=280223800;
   		 PHT_Table[4,38,1]:=63236;
   		 PHT_Table[5,38,0]:=2096853555;
   		 PHT_Table[5,38,1]:=61726;
   		 PHT_Table[0,39,0]:=1804659303;
   		 PHT_Table[0,39,1]:=33594;
   		 PHT_Table[1,39,0]:=-374141133;
   		 PHT_Table[1,39,1]:=20388;
   		 PHT_Table[2,39,0]:=480364209;
   		 PHT_Table[2,39,1]:=52306;
   		 PHT_Table[3,39,0]:=965495713;
   		 PHT_Table[3,39,1]:=33782;
   		 PHT_Table[4,39,0]:=1316092405;
   		 PHT_Table[4,39,1]:=52382;
   		 PHT_Table[5,39,0]:=1215675959;
   		 PHT_Table[5,39,1]:=7608;
   		 PHT_Table[0,40,0]:=-1298803312;
   		 PHT_Table[0,40,1]:=26811;
   		 PHT_Table[1,40,0]:=1356900109;
   		 PHT_Table[1,40,1]:=23555;
   		 PHT_Table[2,40,0]:=1519847407;
   		 PHT_Table[2,40,1]:=13452;
   		 PHT_Table[3,40,0]:=1053770391;
   		 PHT_Table[3,40,1]:=26767;
   		 PHT_Table[4,40,0]:=-688314358;
   		 PHT_Table[4,40,1]:=13496;
   		 PHT_Table[5,40,0]:=-941144045;
   		 PHT_Table[5,40,1]:=53337;
   		 PHT_Table[0,41,0]:=908414410;
   		 PHT_Table[0,41,1]:=20831;
   		 PHT_Table[1,41,0]:=1921827810;
   		 PHT_Table[1,41,1]:=62636;
   		 PHT_Table[2,41,0]:=-1209194586;
   		 PHT_Table[2,41,1]:=42326;
   		 PHT_Table[3,41,0]:=1620222189;
   		 PHT_Table[3,41,1]:=20986;
   		 PHT_Table[4,41,0]:=-503367227;
   		 PHT_Table[4,41,1]:=42483;
   		 PHT_Table[5,41,0]:=-1616157258;
   		 PHT_Table[5,41,1]:=41499;
   		 PHT_Table[0,42,0]:=1853078128;
   		 PHT_Table[0,42,1]:=53609;
   		 PHT_Table[1,42,0]:=816420082;
   		 PHT_Table[1,42,1]:=13313;
   		 PHT_Table[2,42,0]:=914683052;
   		 PHT_Table[2,42,1]:=58765;
   		 PHT_Table[3,42,0]:=-482001276;
   		 PHT_Table[3,42,1]:=53644;
   		 PHT_Table[4,42,0]:=-1151920122;
   		 PHT_Table[4,42,1]:=58728;
   		 PHT_Table[5,42,0]:=-1268958984;
   		 PHT_Table[5,42,1]:=47415;
   		 PHT_Table[0,43,0]:=-254961219;
   		 PHT_Table[0,43,1]:=63945;
   		 PHT_Table[1,43,0]:=1104582135;
   		 PHT_Table[1,43,1]:=2265;
   		 PHT_Table[2,43,0]:=-1582688442;
   		 PHT_Table[2,43,1]:=61921;
   		 PHT_Table[3,43,0]:=292303786;
   		 PHT_Table[3,43,1]:=63800;
   		 PHT_Table[4,43,0]:=1090170336;
   		 PHT_Table[4,43,1]:=61712;
   		 PHT_Table[5,43,0]:=-339618868;
   		 PHT_Table[5,43,1]:=59768;
   		 PHT_Table[0,44,0]:=1080126674;
   		 PHT_Table[0,44,1]:=58021;
   		 PHT_Table[1,44,0]:=-979616809;
   		 PHT_Table[1,44,1]:=37784;
   		 PHT_Table[2,44,0]:=-1200051630;
   		 PHT_Table[2,44,1]:=29004;
   		 PHT_Table[3,44,0]:=215553144;
   		 PHT_Table[3,44,1]:=58068;
   		 PHT_Table[4,44,0]:=-189665411;
   		 PHT_Table[4,44,1]:=28989;
   		 PHT_Table[5,44,0]:=-1120507568;
   		 PHT_Table[5,44,1]:=57120;
   		 PHT_Table[0,45,0]:=-181483094;
   		 PHT_Table[0,45,1]:=43930;
   		 PHT_Table[1,45,0]:=-1731457482;
   		 PHT_Table[1,45,1]:=29564;
   		 PHT_Table[2,45,0]:=-1953553061;
   		 PHT_Table[2,45,1]:=55358;
   		 PHT_Table[3,45,0]:=-878360945;
   		 PHT_Table[3,45,1]:=43842;
   		 PHT_Table[4,45,0]:=-1243853805;
   		 PHT_Table[4,45,1]:=55526;
   		 PHT_Table[5,45,0]:=401167619;
   		 PHT_Table[5,45,1]:=19959;
   		 PHT_Table[0,46,0]:=406297448;
   		 PHT_Table[0,46,1]:=25235;
   		 PHT_Table[1,46,0]:=-2017891129;
   		 PHT_Table[1,46,1]:=21301;
   		 PHT_Table[2,46,0]:=957446488;
   		 PHT_Table[2,46,1]:=12695;
   		 PHT_Table[3,46,0]:=-1894872559;
   		 PHT_Table[3,46,1]:=25250;
   		 PHT_Table[4,46,0]:=-1374040386;
   		 PHT_Table[4,46,1]:=12710;
   		 PHT_Table[5,46,0]:=-1765788642;
   		 PHT_Table[5,46,1]:=50188;
   		 PHT_Table[0,47,0]:=-1137035941;
   		 PHT_Table[0,47,1]:=10920;
   		 PHT_Table[1,47,0]:=1251711182;
   		 PHT_Table[1,47,1]:=16342;
   		 PHT_Table[2,47,0]:=-2007561160;
   		 PHT_Table[2,47,1]:=5483;
   		 PHT_Table[3,47,0]:=-676175273;
   		 PHT_Table[3,47,1]:=10941;
   		 PHT_Table[4,47,0]:=-473291326;
   		 PHT_Table[4,47,1]:=5502;
   		 PHT_Table[5,47,0]:=496476307;
   		 PHT_Table[5,47,1]:=21598;
   		 PHT_Table[0,48,0]:=-2010752914;
   		 PHT_Table[0,48,1]:=2080;
   		 PHT_Table[1,48,0]:=-323137023;
   		 PHT_Table[1,48,1]:=3128;
   		 PHT_Table[2,48,0]:=2097123685;
   		 PHT_Table[2,48,1]:=1052;
   		 PHT_Table[3,48,0]:=-1805998081;
   		 PHT_Table[3,48,1]:=2084;
   		 PHT_Table[4,48,0]:=1619490448;
   		 PHT_Table[4,48,1]:=1048;
   		 PHT_Table[5,48,0]:=321664938;
   		 PHT_Table[5,48,1]:=4164;
   		 PHT_Table[0,49,0]:=105603098;
   		 PHT_Table[0,49,1]:=38242;
   		 PHT_Table[1,49,0]:=1743068023;
   		 PHT_Table[1,49,1]:=21190;
   		 PHT_Table[2,49,0]:=-976235242;
   		 PHT_Table[2,49,1]:=51043;
   		 PHT_Table[3,49,0]:=1703849935;
   		 PHT_Table[3,49,1]:=38309;
   		 PHT_Table[4,49,0]:=-1496465758;
   		 PHT_Table[4,49,1]:=51108;
   		 PHT_Table[5,49,0]:=-1473245814;
   		 PHT_Table[5,49,1]:=12547;
   		 PHT_Table[0,50,0]:=1253887228;
   		 PHT_Table[0,50,1]:=17923;
   		 PHT_Table[1,50,0]:=1822955086;
   		 PHT_Table[1,50,1]:=26057;
   		 PHT_Table[2,50,0]:=-332214680;
   		 PHT_Table[2,50,1]:=9193;
   		 PHT_Table[3,50,0]:=-1554973134;
   		 PHT_Table[3,50,1]:=17952;
   		 PHT_Table[4,50,0]:=100480640;
   		 PHT_Table[4,50,1]:=9162;
   		 PHT_Table[5,50,0]:=1583775445;
   		 PHT_Table[5,50,1]:=35877;
   		 PHT_Table[0,51,0]:=-1905444748;
   		 PHT_Table[0,51,1]:=40258;
   		 PHT_Table[1,51,0]:=-1957148298;
   		 PHT_Table[1,51,1]:=24318;
   		 PHT_Table[2,51,0]:=-1188019085;
   		 PHT_Table[2,51,1]:=50047;
   		 PHT_Table[3,51,0]:=-237762512;
   		 PHT_Table[3,51,1]:=40321;
   		 PHT_Table[4,51,0]:=-968177614;
   		 PHT_Table[4,51,1]:=50108;
   		 PHT_Table[5,51,0]:=-1155778016;
   		 PHT_Table[5,51,1]:=8519;
   		 PHT_Table[0,52,0]:=500484991;
   		 PHT_Table[0,52,1]:=12480;
   		 PHT_Table[1,52,0]:=1587803910;
   		 PHT_Table[1,52,1]:=10384;
   		 PHT_Table[2,52,0]:=322194245;
   		 PHT_Table[2,52,1]:=6216;
   		 PHT_Table[3,52,0]:=1439170356;
   		 PHT_Table[3,52,1]:=12504;
   		 PHT_Table[4,52,0]:=1530867533;
   		 PHT_Table[4,52,1]:=6224;
   		 PHT_Table[5,52,0]:=1793635025;
   		 PHT_Table[5,52,1]:=24707;
   		 PHT_Table[0,53,0]:=1778514581;
   		 PHT_Table[0,53,1]:=14300;
   		 PHT_Table[1,53,0]:=-2082044248;
   		 PHT_Table[1,53,1]:=41349;
   		 PHT_Table[2,53,0]:=-1341220031;
   		 PHT_Table[2,53,1]:=38607;
   		 PHT_Table[3,53,0]:=-1515064306;
   		 PHT_Table[3,53,1]:=14154;
   		 PHT_Table[4,53,0]:=2133380147;
   		 PHT_Table[4,53,1]:=38489;
   		 PHT_Table[5,53,0]:=-1921136643;
   		 PHT_Table[5,53,1]:=28213;
   		 PHT_Table[0,54,0]:=-1432203528;
   		 PHT_Table[0,54,1]:=2600;
   		 PHT_Table[1,54,0]:=-681980982;
   		 PHT_Table[1,54,1]:=3894;
   		 PHT_Table[2,54,0]:=1669758647;
   		 PHT_Table[2,54,1]:=1307;
   		 PHT_Table[3,54,0]:=-1312700282;
   		 PHT_Table[3,54,1]:=2605;
   		 PHT_Table[4,54,0]:=2028005044;
   		 PHT_Table[4,54,1]:=1310;
   		 PHT_Table[5,54,0]:=1361542157;
   		 PHT_Table[5,54,1]:=5205;
   		 PHT_Table[0,55,0]:=-378858969;
   		 PHT_Table[0,55,1]:=12220;
   		 PHT_Table[1,55,0]:=-1405456213;
   		 PHT_Table[1,55,1]:=46541;
   		 PHT_Table[2,55,0]:=873739246;
   		 PHT_Table[2,55,1]:=39659;
   		 PHT_Table[3,55,0]:=39781908;
   		 PHT_Table[3,55,1]:=12070;
   		 PHT_Table[4,55,0]:=-541436264;
   		 PHT_Table[4,55,1]:=39537;
   		 PHT_Table[5,55,0]:=-1207329256;
   		 PHT_Table[5,55,1]:=24313;
   		 PHT_Table[0,56,0]:=-290364721;
   		 PHT_Table[0,56,1]:=3640;
   		 PHT_Table[1,56,0]:=-1584733625;
   		 PHT_Table[1,56,1]:=2346;
   		 PHT_Table[2,56,0]:=1567931144;
   		 PHT_Table[2,56,1]:=1813;
   		 PHT_Table[3,56,0]:=-68413836;
   		 PHT_Table[3,56,1]:=3647;
   		 PHT_Table[4,56,0]:=1211031036;
   		 PHT_Table[4,56,1]:=1810;
   		 PHT_Table[5,56,0]:=-718149032;
   		 PHT_Table[5,56,1]:=7287;
   		 PHT_Table[0,57,0]:=1384863636;
   		 PHT_Table[0,57,1]:=9360;
   		 PHT_Table[1,57,0]:=-351176055;
   		 PHT_Table[1,57,1]:=14076;
   		 PHT_Table[2,57,0]:=-719079632;
   		 PHT_Table[2,57,1]:=4734;
   		 PHT_Table[3,57,0]:=744387619;
   		 PHT_Table[3,57,1]:=9346;
   		 PHT_Table[4,57,0]:=-1411057602;
   		 PHT_Table[4,57,1]:=4716;
   		 PHT_Table[5,57,0]:=-928625973;
   		 PHT_Table[5,57,1]:=18473;
   		 PHT_Table[0,58,0]:=-1330842257;
   		 PHT_Table[0,58,1]:=7020;
   		 PHT_Table[1,58,0]:=-2075480544;
   		 PHT_Table[1,58,1]:=39745;
   		 PHT_Table[2,58,0]:=433241364;
   		 PHT_Table[2,58,1]:=32941;
   		 PHT_Table[3,58,0]:=498411474;
   		 PHT_Table[3,58,1]:=7148;
   		 PHT_Table[4,58,0]:=-1270136163;
   		 PHT_Table[4,58,1]:=32813;
   		 PHT_Table[5,58,0]:=1459075740;
   		 PHT_Table[5,58,1]:=13912;
   		 PHT_Table[0,59,0]:=-2134714177;
   		 PHT_Table[0,59,1]:=57169;
   		 PHT_Table[1,59,0]:=-1859946827;
   		 PHT_Table[1,59,1]:=15659;
   		 PHT_Table[2,59,0]:=1810911140;
   		 PHT_Table[2,59,1]:=58008;
   		 PHT_Table[3,59,0]:=413739248;
   		 PHT_Table[3,59,1]:=57267;
   		 PHT_Table[4,59,0]:=-210123270;
   		 PHT_Table[4,59,1]:=57978;
   		 PHT_Table[5,59,0]:=1634521760;
   		 PHT_Table[5,59,1]:=42304;
   		 PHT_Table[0,60,0]:=-1458929931;
   		 PHT_Table[0,60,1]:=52505;
   		 PHT_Table[1,60,0]:=1772505980;
   		 PHT_Table[1,60,1]:=9813;
   		 PHT_Table[2,60,0]:=-1939039812;
   		 PHT_Table[2,60,1]:=60327;
   		 PHT_Table[3,60,0]:=243667564;
   		 PHT_Table[3,60,1]:=52722;
   		 PHT_Table[4,60,0]:=722188773;
   		 PHT_Table[4,60,1]:=60236;
   		 PHT_Table[5,60,0]:=88078152;
   		 PHT_Table[5,60,1]:=33241;
   		 PHT_Table[0,61,0]:=-1030056814;
   		 PHT_Table[0,61,1]:=20003;
   		 PHT_Table[1,61,0]:=-2146089905;
   		 PHT_Table[1,61,1]:=27121;
   		 PHT_Table[2,61,0]:=-1865588979;
   		 PHT_Table[2,61,1]:=10229;
   		 PHT_Table[3,61,0]:=923425229;
   		 PHT_Table[3,61,1]:=19972;
   		 PHT_Table[4,61,0]:=1702510608;
   		 PHT_Table[4,61,1]:=10194;
   		 PHT_Table[5,61,0]:=1296714111;
   		 PHT_Table[5,61,1]:=40033;
   		 PHT_Table[0,62,0]:=-838052698;
   		 PHT_Table[0,62,1]:=32743;
   		 PHT_Table[1,62,0]:=1321497249;
   		 PHT_Table[1,62,1]:=52582;
   		 PHT_Table[2,62,0]:=21556769;
   		 PHT_Table[2,62,1]:=45619;
   		 PHT_Table[3,62,0]:=-49472440;
   		 PHT_Table[3,62,1]:=32597;
   		 PHT_Table[4,62,0]:=855320399;
   		 PHT_Table[4,62,1]:=45697;
   		 PHT_Table[5,62,0]:=103437168;
   		 PHT_Table[5,62,1]:=65127;
   		 PHT_Table[0,63,0]:=-934857540;
   		 PHT_Table[0,63,1]:=60037;
   		 PHT_Table[1,63,0]:=690055638;
   		 PHT_Table[1,63,1]:=40864;
   		 PHT_Table[2,63,0]:=-997770441;
   		 PHT_Table[2,63,1]:=30032;
   		 PHT_Table[3,63,0]:=-1736199289;
   		 PHT_Table[3,63,1]:=60144;
   		 PHT_Table[4,63,0]:=-1808360979;
   		 PHT_Table[4,63,1]:=29989;
   		 PHT_Table[5,63,0]:=-1374003462;
   		 PHT_Table[5,63,1]:=53092;
   		 PHT_Table[0,64,0]:=701015626;
   		 PHT_Table[0,64,1]:=4680;
   		 PHT_Table[1,64,0]:=-125485623;
   		 PHT_Table[1,64,1]:=7038;
   		 PHT_Table[2,64,0]:=-409151976;
   		 PHT_Table[2,64,1]:=2367;
   		 PHT_Table[3,64,0]:=372193948;
   		 PHT_Table[3,64,1]:=4673;
   		 PHT_Table[4,64,0]:=-663585761;
   		 PHT_Table[4,64,1]:=2358;
   		 PHT_Table[5,64,0]:=1683170792;
   		 PHT_Table[5,64,1]:=9369;
   		 PHT_Table[0,65,0]:=-700723250;
   		 PHT_Table[0,65,1]:=7540;
   		 PHT_Table[1,65,0]:=-914547098;
   		 PHT_Table[1,65,1]:=40531;
   		 PHT_Table[2,65,0]:=945395577;
   		 PHT_Table[2,65,1]:=33700;
   		 PHT_Table[3,65,0]:=1912837721;
   		 PHT_Table[3,65,1]:=7671;
   		 PHT_Table[4,65,0]:=-1662850575;
   		 PHT_Table[4,65,1]:=33575;
   		 PHT_Table[5,65,0]:=-1863686290;
   		 PHT_Table[5,65,1]:=14955;
   		 PHT_Table[0,66,0]:=-1354686737;
   		 PHT_Table[0,66,1]:=22651;
   		 PHT_Table[1,66,0]:=239292427;
   		 PHT_Table[1,66,1]:=29843;
   		 PHT_Table[2,66,0]:=1235438762;
   		 PHT_Table[2,66,1]:=11460;
   		 PHT_Table[3,66,0]:=1795734947;
   		 PHT_Table[3,66,1]:=22615;
   		 PHT_Table[4,66,0]:=-1916401849;
   		 PHT_Table[4,66,1]:=11496;
   		 PHT_Table[5,66,0]:=-1391461694;
   		 PHT_Table[5,66,1]:=45274;
   		 PHT_Table[0,67,0]:=1506273096;
   		 PHT_Table[0,67,1]:=13520;
   		 PHT_Table[1,67,0]:=678485643;
   		 PHT_Table[1,67,1]:=11916;
   		 PHT_Table[2,67,0]:=767987450;
   		 PHT_Table[2,67,1]:=6726;
   		 PHT_Table[3,67,0]:=535437766;
   		 PHT_Table[3,67,1]:=13514;
   		 PHT_Table[4,67,0]:=1810961413;
   		 PHT_Table[4,67,1]:=6748;
   		 PHT_Table[5,67,0]:=-285334396;
   		 PHT_Table[5,67,1]:=26785;
   		 PHT_Table[0,68,0]:=2068050398;
   		 PHT_Table[0,68,1]:=14040;
   		 PHT_Table[1,68,0]:=328484672;
   		 PHT_Table[1,68,1]:=11650;
   		 PHT_Table[2,68,0]:=851403048;
   		 PHT_Table[2,68,1]:=6977;
   		 PHT_Table[3,68,0]:=980504255;
   		 PHT_Table[3,68,1]:=14019;
   		 PHT_Table[4,68,0]:=1939244065;
   		 PHT_Table[4,68,1]:=7002;
   		 PHT_Table[5,68,0]:=-1393201373;
   		 PHT_Table[5,68,1]:=27824;
   		 PHT_Table[0,69,0]:=-1291532958;
   		 PHT_Table[0,69,1]:=56413;
   		 PHT_Table[1,69,0]:=984952470;
   		 PHT_Table[1,69,1]:=45602;
   		 PHT_Table[2,69,0]:=-164079073;
   		 PHT_Table[2,69,1]:=28177;
   		 PHT_Table[3,69,0]:=-1561133768;
   		 PHT_Table[3,69,1]:=56371;
   		 PHT_Table[4,69,0]:=-408937012;
   		 PHT_Table[4,69,1]:=28287;
   		 PHT_Table[5,69,0]:=49230297;
   		 PHT_Table[5,69,1]:=41940;
   		 PHT_Table[0,70,0]:=26284274;
   		 PHT_Table[0,70,1]:=46310;
   		 PHT_Table[1,70,0]:=1783990683;
   		 PHT_Table[1,70,1]:=60961;
   		 PHT_Table[2,70,0]:=-1397793296;
   		 PHT_Table[2,70,1]:=23197;
   		 PHT_Table[3,70,0]:=-1673674833;
   		 PHT_Table[3,70,1]:=46268;
   		 PHT_Table[4,70,0]:=827930054;
   		 PHT_Table[4,70,1]:=23239;
   		 PHT_Table[5,70,0]:=-989300278;
   		 PHT_Table[5,70,1]:=29581;
   		 PHT_Table[0,71,0]:=-1668873422;
   		 PHT_Table[0,71,1]:=23415;
   		 PHT_Table[1,71,0]:=-1512765400;
   		 PHT_Table[1,71,1]:=64410;
   		 PHT_Table[2,71,0]:=-731162351;
   		 PHT_Table[2,71,1]:=41037;
   		 PHT_Table[3,71,0]:=-783062933;
   		 PHT_Table[3,71,1]:=23511;
   		 PHT_Table[4,71,0]:=-1725964431;
   		 PHT_Table[4,71,1]:=41197;
   		 PHT_Table[5,71,0]:=-829679173;
   		 PHT_Table[5,71,1]:=46670;
   		 PHT_Table[0,72,0]:=182296622;
   		 PHT_Table[0,72,1]:=42150;
   		 PHT_Table[1,72,0]:=-1456198247;
   		 PHT_Table[1,72,1]:=63057;
   		 PHT_Table[2,72,0]:=1414161466;
   		 PHT_Table[2,72,1]:=21157;
   		 PHT_Table[3,72,0]:=-1349916086;
   		 PHT_Table[3,72,1]:=42228;
   		 PHT_Table[4,72,0]:=-246621699;
   		 PHT_Table[4,72,1]:=21239;
   		 PHT_Table[5,72,0]:=-481290363;
   		 PHT_Table[5,72,1]:=21253;
   		 PHT_Table[0,73,0]:=1466435459;
   		 PHT_Table[0,73,1]:=30403;
   		 PHT_Table[1,73,0]:=839639368;
   		 PHT_Table[1,73,1]:=19801;
   		 PHT_Table[2,73,0]:=-16349907;
   		 PHT_Table[2,73,1]:=15265;
   		 PHT_Table[3,73,0]:=-157875962;
   		 PHT_Table[3,73,1]:=30456;
   		 PHT_Table[4,73,0]:=1589778893;
   		 PHT_Table[4,73,1]:=15258;
   		 PHT_Table[5,73,0]:=881773572;
   		 PHT_Table[5,73,1]:=60582;
   		 PHT_Table[0,74,0]:=844565807;
   		 PHT_Table[0,74,1]:=47082;
   		 PHT_Table[1,74,0]:=-1044131400;
   		 PHT_Table[1,74,1]:=24872;
   		 PHT_Table[2,74,0]:=828852299;
   		 PHT_Table[2,74,1]:=54804;
   		 PHT_Table[3,74,0]:=644246119;
   		 PHT_Table[3,74,1]:=46908;
   		 PHT_Table[4,74,0]:=629206512;
   		 PHT_Table[4,74,1]:=54978;
   		 PHT_Table[5,74,0]:=-1500800333;
   		 PHT_Table[5,74,1]:=29977;
   		 PHT_Table[0,75,0]:=-326614480;
   		 PHT_Table[0,75,1]:=32239;
   		 PHT_Table[1,75,0]:=1965091690;
   		 PHT_Table[1,75,1]:=52840;
   		 PHT_Table[2,75,0]:=506528243;
   		 PHT_Table[2,75,1]:=45876;
   		 PHT_Table[3,75,0]:=-661228751;
   		 PHT_Table[3,75,1]:=32092;
   		 PHT_Table[4,75,0]:=714913643;
   		 PHT_Table[4,75,1]:=45959;
   		 PHT_Table[5,75,0]:=1143019735;
   		 PHT_Table[5,75,1]:=64118;
   		 PHT_Table[0,76,0]:=98783255;
   		 PHT_Table[0,76,1]:=21075;
   		 PHT_Table[1,76,0]:=-652567615;
   		 PHT_Table[1,76,1]:=31653;
   		 PHT_Table[2,76,0]:=707080733;
   		 PHT_Table[2,76,1]:=10719;
   		 PHT_Table[3,76,0]:=-624331483;
   		 PHT_Table[3,76,1]:=21114;
   		 PHT_Table[4,76,0]:=-182001165;
   		 PHT_Table[4,76,1]:=10742;
   		 PHT_Table[5,76,0]:=-64452913;
   		 PHT_Table[5,76,1]:=42127;
   		 PHT_Table[0,77,0]:=-1572418007;
   		 PHT_Table[0,77,1]:=56665;
   		 PHT_Table[1,77,0]:=-1429737602;
   		 PHT_Table[1,77,1]:=15909;
   		 PHT_Table[2,77,0]:=1955176566;
   		 PHT_Table[2,77,1]:=58271;
   		 PHT_Table[3,77,0]:=1026705289;
   		 PHT_Table[3,77,1]:=56762;
   		 PHT_Table[4,77,0]:=-350333474;
   		 PHT_Table[4,77,1]:=58236;
   		 PHT_Table[5,77,0]:=593991943;
   		 PHT_Table[5,77,1]:=41297;
   		 PHT_Table[0,78,0]:=-908712882;
   		 PHT_Table[0,78,1]:=24163;
   		 PHT_Table[1,78,0]:=1131733069;
   		 PHT_Table[1,78,1]:=29057;
   		 PHT_Table[2,78,0]:=1747478215;
   		 PHT_Table[2,78,1]:=12237;
   		 PHT_Table[3,78,0]:=79563816;
   		 PHT_Table[3,78,1]:=24140;
   		 PHT_Table[4,78,0]:=-1519408085;
   		 PHT_Table[4,78,1]:=12258;
   		 PHT_Table[5,78,0]:=1796351792;
   		 PHT_Table[5,78,1]:=48361;
   		 PHT_Table[0,79,0]:=948612353;
   		 PHT_Table[0,79,1]:=4940;
   		 PHT_Table[1,79,0]:=1761082401;
   		 PHT_Table[1,79,1]:=38777;
   		 PHT_Table[2,79,0]:=1697459313;
   		 PHT_Table[2,79,1]:=33969;
   		 PHT_Table[3,79,0]:=-1980792787;
   		 PHT_Table[3,79,1]:=5064;
   		 PHT_Table[4,79,0]:=-724814835;
   		 PHT_Table[4,79,1]:=33845;
   		 PHT_Table[5,79,0]:=1172016438;
   		 PHT_Table[5,79,1]:=9756;
   		 PHT_Table[0,80,0]:=676968120;
   		 PHT_Table[0,80,1]:=42670;
   		 PHT_Table[1,80,0]:=-1831816110;
   		 PHT_Table[1,80,1]:=62815;
   		 PHT_Table[2,80,0]:=1261669352;
   		 PHT_Table[2,80,1]:=21410;
   		 PHT_Table[3,80,0]:=-1978497741;
   		 PHT_Table[3,80,1]:=42749;
   		 PHT_Table[4,80,0]:=-383039015;
   		 PHT_Table[4,80,1]:=21489;
   		 PHT_Table[5,80,0]:=-1587848158;
   		 PHT_Table[5,80,1]:=22292;
   		 PHT_Table[0,81,0]:=-588877856;
   		 PHT_Table[0,81,1]:=47570;
   		 PHT_Table[1,81,0]:=1615410175;
   		 PHT_Table[1,81,1]:=26626;
   		 PHT_Table[2,81,0]:=1813246787;
   		 PHT_Table[2,81,1]:=53505;
   		 PHT_Table[3,81,0]:=-578126829;
   		 PHT_Table[3,81,1]:=47363;
   		 PHT_Table[4,81,0]:=1840132108;
   		 PHT_Table[4,81,1]:=53712;
   		 PHT_Table[5,81,0]:=1941598443;
   		 PHT_Table[5,81,1]:=26990;
   		 PHT_Table[0,82,0]:=0;
   		 PHT_Table[0,82,1]:=0;
   		 PHT_Table[1,82,0]:=0;
   		 PHT_Table[1,82,1]:=0;
   		 PHT_Table[2,82,0]:=0;
   		 PHT_Table[2,82,1]:=0;
   		 PHT_Table[3,82,0]:=0;
   		 PHT_Table[3,82,1]:=0;
   		 PHT_Table[4,82,0]:=0;
   		 PHT_Table[4,82,1]:=0;
   		 PHT_Table[5,82,0]:=0;
   		 PHT_Table[5,82,1]:=0;
   		 PHT_Table[0,83,0]:=1698630316;
   		 PHT_Table[0,83,1]:=49449;
   		 PHT_Table[1,83,0]:=-204984080;
   		 PHT_Table[1,83,1]:=11377;
   		 PHT_Table[2,83,0]:=-832451226;
   		 PHT_Table[2,83,1]:=60853;
   		 PHT_Table[3,83,0]:=-789484703;
   		 PHT_Table[3,83,1]:=49604;
   		 PHT_Table[4,83,0]:=2067985469;
   		 PHT_Table[4,83,1]:=60760;
   		 PHT_Table[5,83,0]:=-1845143881;
   		 PHT_Table[5,83,1]:=39359;
   		 PHT_Table[0,84,0]:=741078621;
   		 PHT_Table[0,84,1]:=16411;
   		 PHT_Table[1,84,0]:=564110856;
   		 PHT_Table[1,84,1]:=24795;
   		 PHT_Table[2,84,0]:=-843455483;
   		 PHT_Table[2,84,1]:=8416;
   		 PHT_Table[3,84,0]:=-857321543;
   		 PHT_Table[3,84,1]:=16443;
   		 PHT_Table[4,84,0]:=760520172;
   		 PHT_Table[4,84,1]:=8384;
   		 PHT_Table[5,84,0]:=-1736727769;
   		 PHT_Table[5,84,1]:=32790;
   		 PHT_Table[0,85,0]:=1361274777;
   		 PHT_Table[0,85,1]:=58273;
   		 PHT_Table[1,85,0]:=1441724991;
   		 PHT_Table[1,85,1]:=8095;
   		 PHT_Table[2,85,0]:=986271803;
   		 PHT_Table[2,85,1]:=64706;
   		 PHT_Table[3,85,0]:=-1827033399;
   		 PHT_Table[3,85,1]:=58205;
   		 PHT_Table[4,85,0]:=-133191825;
   		 PHT_Table[4,85,1]:=64574;
   		 PHT_Table[5,85,0]:=-1665220210;
   		 PHT_Table[5,85,1]:=56741;
   		 PHT_Table[0,86,0]:=-1466208761;
   		 PHT_Table[0,86,1]:=31231;
   		 PHT_Table[1,86,0]:=66306791;
   		 PHT_Table[1,86,1]:=51316;
   		 PHT_Table[2,86,0]:=549700684;
   		 PHT_Table[2,86,1]:=45370;
   		 PHT_Table[3,86,0]:=-1833194045;
   		 PHT_Table[3,86,1]:=31054;
   		 PHT_Table[4,86,0]:=441617443;
   		 PHT_Table[4,86,1]:=45451;
   		 PHT_Table[5,86,0]:=-1070100862;
   		 PHT_Table[5,86,1]:=62036;
   		 PHT_Table[0,87,0]:=588580452;
   		 PHT_Table[0,87,1]:=46830;
   		 PHT_Table[1,87,0]:=1370558544;
   		 PHT_Table[1,87,1]:=60719;
   		 PHT_Table[2,87,0]:=-1277775326;
   		 PHT_Table[2,87,1]:=23450;
   		 PHT_Table[3,87,0]:=-1180249898;
   		 PHT_Table[3,87,1]:=46773;
   		 PHT_Table[4,87,0]:=691971554;
   		 PHT_Table[4,87,1]:=23489;
   		 PHT_Table[5,87,0]:=-2029833619;
   		 PHT_Table[5,87,1]:=30620;
   		 PHT_Table[0,88,0]:=992124172;
   		 PHT_Table[0,88,1]:=54397;
   		 PHT_Table[1,88,0]:=-704086889;
   		 PHT_Table[1,88,1]:=48666;
   		 PHT_Table[2,88,0]:=-1966617734;
   		 PHT_Table[2,88,1]:=27149;
   		 PHT_Table[3,88,0]:=917002951;
   		 PHT_Table[3,88,1]:=54295;
   		 PHT_Table[4,88,0]:=-2027459748;
   		 PHT_Table[4,88,1]:=27239;
   		 PHT_Table[5,88,0]:=297993843;
   		 PHT_Table[5,88,1]:=45968;
   		 PHT_Table[0,89,0]:=-2061399896;
   		 PHT_Table[0,89,1]:=36098;
   		 PHT_Table[1,89,0]:=1211755892;
   		 PHT_Table[1,89,1]:=18062;
   		 PHT_Table[2,89,0]:=1104510393;
   		 PHT_Table[2,89,1]:=52039;
   		 PHT_Table[3,89,0]:=-1033871915;
   		 PHT_Table[3,89,1]:=36297;
   		 PHT_Table[4,89,0]:=106898441;
   		 PHT_Table[4,89,1]:=52108;
   		 PHT_Table[5,89,0]:=-1656466321;
   		 PHT_Table[5,89,1]:=463;
   		 PHT_Table[0,90,0]:=1298578452;
   		 PHT_Table[0,90,1]:=26503;
   		 PHT_Table[1,90,0]:=1628996770;
   		 PHT_Table[1,90,1]:=55598;
   		 PHT_Table[2,90,0]:=-2058205554;
   		 PHT_Table[2,90,1]:=48663;
   		 PHT_Table[3,90,0]:=1524887122;
   		 PHT_Table[3,90,1]:=26425;
   		 PHT_Table[4,90,0]:=-1838563868;
   		 PHT_Table[4,90,1]:=48809;
   		 PHT_Table[5,90,0]:=861801109;
   		 PHT_Table[5,90,1]:=52907;
   		 PHT_Table[0,91,0]:=326839220;
   		 PHT_Table[0,91,1]:=29395;
   		 PHT_Table[1,91,0]:=1155057861;
   		 PHT_Table[1,91,1]:=19269;
   		 PHT_Table[2,91,0]:=-1040957294;
   		 PHT_Table[2,91,1]:=14767;
   		 PHT_Table[3,91,0]:=-1128603660;
   		 PHT_Table[3,91,1]:=29418;
   		 PHT_Table[4,91,0]:=1846289029;
   		 PHT_Table[4,91,1]:=14742;
   		 PHT_Table[5,91,0]:=-1332192687;
   		 PHT_Table[5,91,1]:=58500;
   		 PHT_Table[0,92,0]:=386493265;
   		 PHT_Table[0,92,1]:=37990;
   		 PHT_Table[1,92,0]:=-141043041;
   		 PHT_Table[1,92,1]:=57025;
   		 PHT_Table[2,92,0]:=1199452031;
   		 PHT_Table[2,92,1]:=19181;
   		 PHT_Table[3,92,0]:=-95545986;
   		 PHT_Table[3,92,1]:=37932;
   		 PHT_Table[4,92,0]:=-1435240784;
   		 PHT_Table[4,92,1]:=19111;
   		 PHT_Table[5,92,0]:=-1984387756;
   		 PHT_Table[5,92,1]:=13190;
   		 PHT_Table[0,93,0]:=-616816888;
   		 PHT_Table[0,93,1]:=38998;
   		 PHT_Table[1,93,0]:=1845076243;
   		 PHT_Table[1,93,1]:=54501;
   		 PHT_Table[2,93,0]:=91454373;
   		 PHT_Table[2,93,1]:=19711;
   		 PHT_Table[3,93,0]:=607743091;
   		 PHT_Table[3,93,1]:=38938;
   		 PHT_Table[4,93,0]:=-96814232;
   		 PHT_Table[4,93,1]:=19635;
   		 PHT_Table[5,93,0]:=511837355;
   		 PHT_Table[5,93,1]:=11232;
   		 PHT_Table[0,94,0]:=1166163141;
   		 PHT_Table[0,94,1]:=45302;
   		 PHT_Table[1,94,0]:=478584854;
   		 PHT_Table[1,94,1]:=59453;
   		 PHT_Table[2,94,0]:=-1839359921;
   		 PHT_Table[2,94,1]:=22675;
   		 PHT_Table[3,94,0]:=-703569571;
   		 PHT_Table[3,94,1]:=45230;
   		 PHT_Table[4,94,0]:=26676878;
   		 PHT_Table[4,94,1]:=22731;
   		 PHT_Table[5,94,0]:=1092546463;
   		 PHT_Table[5,94,1]:=31663;
   		 PHT_Table[0,95,0]:=218616006;
   		 PHT_Table[0,95,1]:=34082;
   		 PHT_Table[1,95,0]:=-1534804107;
   		 PHT_Table[1,95,1]:=19126;
   		 PHT_Table[2,95,0]:=1026223324;
   		 PHT_Table[2,95,1]:=53083;
   		 PHT_Table[3,95,0]:=1446705706;
   		 PHT_Table[3,95,1]:=34285;
   		 PHT_Table[4,95,0]:=1725452953;
   		 PHT_Table[4,95,1]:=53140;
   		 PHT_Table[5,95,0]:=-1905761339;
   		 PHT_Table[5,95,1]:=4491;
   		 PHT_Table[0,96,0]:=-27100810;
   		 PHT_Table[0,96,1]:=48090;
   		 PHT_Table[1,96,0]:=1538107956;
   		 PHT_Table[1,96,1]:=27404;
   		 PHT_Table[2,96,0]:=1936333969;
   		 PHT_Table[2,96,1]:=53254;
   		 PHT_Table[3,96,0]:=-133098646;
   		 PHT_Table[3,96,1]:=47882;
   		 PHT_Table[4,96,0]:=1976148008;
   		 PHT_Table[4,96,1]:=53462;
   		 PHT_Table[5,96,0]:=833698636;
   		 PHT_Table[5,96,1]:=28031;
   		 PHT_Table[0,97,0]:=556541595;
   		 PHT_Table[0,97,1]:=50489;
   		 PHT_Table[1,97,0]:=-2061821571;
   		 PHT_Table[1,97,1]:=10861;
   		 PHT_Table[2,97,0]:=-258799399;
   		 PHT_Table[2,97,1]:=61371;
   		 PHT_Table[3,97,0]:=-1696811629;
   		 PHT_Table[3,97,1]:=50646;
   		 PHT_Table[4,97,0]:=1267519349;
   		 PHT_Table[4,97,1]:=61268;
   		 PHT_Table[5,97,0]:=370393314;
   		 PHT_Table[5,97,1]:=37277;
   		 PHT_Table[0,98,0]:=-740778023;
   		 PHT_Table[0,98,1]:=20263;
   		 PHT_Table[1,98,0]:=275219879;
   		 PHT_Table[1,98,1]:=58870;
   		 PHT_Table[2,98,0]:=310158692;
   		 PHT_Table[2,98,1]:=43643;
   		 PHT_Table[3,98,0]:=-1463098500;
   		 PHT_Table[3,98,1]:=20365;
   		 PHT_Table[4,98,0]:=1774454786;
   		 PHT_Table[4,98,1]:=43729;
   		 PHT_Table[5,98,0]:=1824711073;
   		 PHT_Table[5,98,1]:=40676;
   		 PHT_Table[0,99,0]:=-1080949418;
   		 PHT_Table[0,99,1]:=60825;
   		 PHT_Table[1,99,0]:=-194766728;
   		 PHT_Table[1,99,1]:=5813;
   		 PHT_Table[2,99,0]:=1740499763;
   		 PHT_Table[2,99,1]:=64471;
   		 PHT_Table[3,99,0]:=1760934077;
   		 PHT_Table[3,99,1]:=60770;
   		 PHT_Table[4,99,0]:=-1339983213;
   		 PHT_Table[4,99,1]:=64300;
   		 PHT_Table[5,99,0]:=1234119638;
   		 PHT_Table[5,99,1]:=49618;
   		 PHT_Table[0,100,0]:=1052888347;
   		 PHT_Table[0,100,1]:=34350;
   		 PHT_Table[1,100,0]:=252897110;
   		 PHT_Table[1,100,1]:=50623;
   		 PHT_Table[2,100,0]:=-1595737753;
   		 PHT_Table[2,100,1]:=17362;
   		 PHT_Table[3,100,0]:=-329175070;
   		 PHT_Table[3,100,1]:=34413;
   		 PHT_Table[4,100,0]:=1912703663;
   		 PHT_Table[4,100,1]:=17297;
   		 PHT_Table[5,100,0]:=-303333188;
   		 PHT_Table[5,100,1]:=5919;
   		 PHT_Table[0,101,0]:=-105379426;
   		 PHT_Table[0,101,1]:=39518;
   		 PHT_Table[1,101,0]:=1444755672;
   		 PHT_Table[1,101,1]:=55275;
   		 PHT_Table[2,101,0]:=436900983;
   		 PHT_Table[2,101,1]:=19960;
   		 PHT_Table[3,101,0]:=27394826;
   		 PHT_Table[3,101,1]:=39443;
   		 PHT_Table[4,101,0]:=-497210548;
   		 PHT_Table[4,101,1]:=19893;
   		 PHT_Table[5,101,0]:=1552502540;
   		 PHT_Table[5,101,1]:=12273;
   		 PHT_Table[0,102,0]:=1545910111;
   		 PHT_Table[0,102,1]:=26243;
   		 PHT_Table[1,102,0]:=-244693686;
   		 PHT_Table[1,102,1]:=21801;
   		 PHT_Table[2,102,0]:=132365543;
   		 PHT_Table[2,102,1]:=13209;
   		 PHT_Table[3,102,0]:=-987540253;
   		 PHT_Table[3,102,1]:=26288;
   		 PHT_Table[4,102,0]:=-1630013962;
   		 PHT_Table[4,102,1]:=13226;
   		 PHT_Table[5,102,0]:=316056139;
   		 PHT_Table[5,102,1]:=52270;
   		 PHT_Table[0,103,0]:=437173143;
   		 PHT_Table[0,103,1]:=4420;
   		 PHT_Table[1,103,0]:=1393780202;
   		 PHT_Table[1,103,1]:=38007;
   		 PHT_Table[2,103,0]:=2052375459;
   		 PHT_Table[2,103,1]:=34230;
   		 PHT_Table[3,103,0]:=-1401622700;
   		 PHT_Table[3,103,1]:=4545;
   		 PHT_Table[4,103,0]:=-861166551;
   		 PHT_Table[4,103,1]:=34099;
   		 PHT_Table[5,103,0]:=131122833;
   		 PHT_Table[5,103,1]:=8717;
   		 PHT_Table[0,104,0]:=-218842814;
   		 PHT_Table[0,104,1]:=35358;
   		 PHT_Table[1,104,0]:=-1786995494;
   		 PHT_Table[1,104,1]:=53147;
   		 PHT_Table[2,104,0]:=-487608899;
   		 PHT_Table[2,104,1]:=17856;
   		 PHT_Table[3,104,0]:=840324847;
   		 PHT_Table[3,104,1]:=35419;
   		 PHT_Table[4,104,0]:=575194999;
   		 PHT_Table[4,104,1]:=17797;
   		 PHT_Table[5,104,0]:=2060525891;
   		 PHT_Table[5,104,1]:=3961;
   		 PHT_Table[0,105,0]:=-75421343;
   		 PHT_Table[0,105,1]:=59785;
   		 PHT_Table[1,105,0]:=-2101923339;
   		 PHT_Table[1,105,1]:=4265;
   		 PHT_Table[2,105,0]:=1498361484;
   		 PHT_Table[2,105,1]:=63961;
   		 PHT_Table[3,105,0]:=584607311;
   		 PHT_Table[3,105,1]:=59760;
   		 PHT_Table[4,105,0]:=-2131803685;
   		 PHT_Table[4,105,1]:=63776;
   		 PHT_Table[5,105,0]:=-845562493;
   		 PHT_Table[5,105,1]:=51696;
   		 PHT_Table[0,106,0]:=1142107191;
   		 PHT_Table[0,106,1]:=1040;
   		 PHT_Table[1,106,0]:=1993550221;
   		 PHT_Table[1,106,1]:=1564;
   		 PHT_Table[2,106,0]:=1056097727;
   		 PHT_Table[2,106,1]:=526;
   		 PHT_Table[3,106,0]:=1244520178;
   		 PHT_Table[3,106,1]:=1042;
   		 PHT_Table[4,106,0]:=818821960;
   		 PHT_Table[4,106,1]:=524;
   		 PHT_Table[5,106,0]:=-2078894507;
   		 PHT_Table[5,106,1]:=2082;
   		 PHT_Table[0,107,0]:=-2028427177;
   		 PHT_Table[0,107,1]:=65237;
   		 PHT_Table[1,107,0]:=-1668029351;
   		 PHT_Table[1,107,1]:=33228;
   		 PHT_Table[2,107,0]:=43042626;
   		 PHT_Table[2,107,1]:=32614;
   		 PHT_Table[3,107,0]:=-518375280;
   		 PHT_Table[3,107,1]:=65194;
   		 PHT_Table[4,107,0]:=1693273758;
   		 PHT_Table[4,107,1]:=32537;
   		 PHT_Table[5,107,0]:=206874336;
   		 PHT_Table[5,107,1]:=59342;
   		 PHT_Table[0,108,0]:=1322159129;
   		 PHT_Table[0,108,1]:=41142;
   		 PHT_Table[1,108,0]:=-538508268;
   		 PHT_Table[1,108,1]:=61517;
   		 PHT_Table[2,108,0]:=1790484869;
   		 PHT_Table[2,108,1]:=20651;
   		 PHT_Table[3,108,0]:=-442223432;
   		 PHT_Table[3,108,1]:=41190;
   		 PHT_Table[4,108,0]:=-1048386891;
   		 PHT_Table[4,108,1]:=20731;
   		 PHT_Table[5,108,0]:=1732674000;
   		 PHT_Table[5,108,1]:=23335;
   		 PHT_Table[0,109,0]:=-1176935092;
   		 PHT_Table[0,109,1]:=30971;
   		 PHT_Table[1,109,0]:=-1820261617;
   		 PHT_Table[1,109,1]:=17523;
   		 PHT_Table[2,109,0]:=-1569571291;
   		 PHT_Table[2,109,1]:=15540;
   		 PHT_Table[3,109,0]:=226170738;
   		 PHT_Table[3,109,1]:=30919;
   		 PHT_Table[4,109,0]:=384615473;
   		 PHT_Table[4,109,1]:=15496;
   		 PHT_Table[5,109,0]:=-507566500;
   		 PHT_Table[5,109,1]:=61649;
   		 PHT_Table[0,110,0]:=1137269983;
   		 PHT_Table[0,110,1]:=9620;
   		 PHT_Table[1,110,0]:=2070133601;
   		 PHT_Table[1,110,1]:=47867;
   		 PHT_Table[2,110,0]:=1469205849;
   		 PHT_Table[2,110,1]:=40944;
   		 PHT_Table[3,110,0]:=-1281438062;
   		 PHT_Table[3,110,1]:=9483;
   		 PHT_Table[4,110,0]:=-1487228884;
   		 PHT_Table[4,110,1]:=40815;
   		 PHT_Table[5,110,0]:=-382803435;
   		 PHT_Table[5,110,1]:=19116;
   		 PHT_Table[0,111,0]:=-1748257810;
   		 PHT_Table[0,111,1]:=19255;
   		 PHT_Table[1,111,0]:=1723116586;
   		 PHT_Table[1,111,1]:=58346;
   		 PHT_Table[2,111,0]:=747528411;
   		 PHT_Table[2,111,1]:=43125;
   		 PHT_Table[3,111,0]:=-488161906;
   		 PHT_Table[3,111,1]:=19359;
   		 PHT_Table[4,111,0]:=1493840714;
   		 PHT_Table[4,111,1]:=43229;
   		 PHT_Table[5,111,0]:=-388728844;
   		 PHT_Table[5,111,1]:=38598;
   		 PHT_Table[0,112,0]:=1816828559;
   		 PHT_Table[0,112,1]:=41662;
   		 PHT_Table[1,112,0]:=-469525025;
   		 PHT_Table[1,112,1]:=62275;
   		 PHT_Table[2,112,0]:=1975602775;
   		 PHT_Table[2,112,1]:=20908;
   		 PHT_Table[3,112,0]:=-1069589567;
   		 PHT_Table[3,112,1]:=41711;
   		 PHT_Table[4,112,0]:=-639274351;
   		 PHT_Table[4,112,1]:=20989;
   		 PHT_Table[5,112,0]:=625855095;
   		 PHT_Table[5,112,1]:=24374;
   		 PHT_Table[0,113,0]:=-99599981;
   		 PHT_Table[0,113,1]:=23919;
   		 PHT_Table[1,113,0]:=-387794834;
   		 PHT_Table[1,113,1]:=65160;
   		 PHT_Table[2,113,0]:=-169839748;
   		 PHT_Table[2,113,1]:=41796;
   		 PHT_Table[3,113,0]:=-1092232736;
   		 PHT_Table[3,113,1]:=24012;
   		 PHT_Table[4,113,0]:=-1313442787;
   		 PHT_Table[4,113,1]:=41959;
   		 PHT_Table[5,113,0]:=143770697;
   		 PHT_Table[5,113,1]:=47741;
   		 PHT_Table[0,114,0]:=1482094522;
   		 PHT_Table[0,114,1]:=32822;
   		 PHT_Table[1,114,0]:=1109743376;
   		 PHT_Table[1,114,1]:=49325;
   		 PHT_Table[2,114,0]:=-2123771126;
   		 PHT_Table[2,114,1]:=16603;
   		 PHT_Table[3,114,0]:=-2083021207;
   		 PHT_Table[3,114,1]:=32886;
   		 PHT_Table[4,114,0]:=1520968131;
   		 PHT_Table[4,114,1]:=16539;
   		 PHT_Table[5,114,0]:=737566030;
   		 PHT_Table[5,114,1]:=6956;
   		 PHT_Table[0,115,0]:=1431381884;
   		 PHT_Table[0,115,1]:=1300;
   		 PHT_Table[1,115,0]:=-425596827;
   		 PHT_Table[1,115,1]:=35355;
   		 PHT_Table[2,115,0]:=-1136443434;
   		 PHT_Table[2,115,1]:=36736;
   		 PHT_Table[3,115,0]:=-705862589;
   		 PHT_Table[3,115,1]:=1435;
   		 PHT_Table[4,115,0]:=1014002522;
   		 PHT_Table[4,115,1]:=36623;
   		 PHT_Table[5,115,0]:=-1516355957;
   		 PHT_Table[5,115,1]:=2727;
   		 PHT_Table[0,116,0]:=-500718853;
   		 PHT_Table[0,116,1]:=16380;
   		 PHT_Table[1,116,0]:=1868289193;
   		 PHT_Table[1,116,1]:=44477;
   		 PHT_Table[2,116,0]:=-856618460;
   		 PHT_Table[2,116,1]:=37587;
   		 PHT_Table[3,116,0]:=837506033;
   		 PHT_Table[3,116,1]:=16238;
   		 PHT_Table[4,116,0]:=531610275;
   		 PHT_Table[4,116,1]:=37441;
   		 PHT_Table[5,116,0]:=-1638797225;
   		 PHT_Table[5,116,1]:=32369;
   		 PHT_Table[0,117,0]:=131756264;
   		 PHT_Table[0,117,1]:=8580;
   		 PHT_Table[1,117,0]:=229675756;
   		 PHT_Table[1,117,1]:=48359;
   		 PHT_Table[2,117,0]:=1767934182;
   		 PHT_Table[2,117,1]:=40446;
   		 PHT_Table[3,117,0]:=-105705376;
   		 PHT_Table[3,117,1]:=8473;
   		 PHT_Table[4,117,0]:=-1751872668;
   		 PHT_Table[4,117,1]:=40291;
   		 PHT_Table[5,117,0]:=1832416320;
   		 PHT_Table[5,117,1]:=17038;
   		 PHT_Table[0,118,0]:=838810914;
   		 PHT_Table[0,118,1]:=28891;
   		 PHT_Table[1,118,0]:=2134659342;
   		 PHT_Table[1,118,1]:=18507;
   		 PHT_Table[2,118,0]:=-561139904;
   		 PHT_Table[2,118,1]:=14504;
   		 PHT_Table[3,118,0]:=-1725845363;
   		 PHT_Table[3,118,1]:=28899;
   		 PHT_Table[4,118,0]:=1986769569;
   		 PHT_Table[4,118,1]:=14480;
   		 PHT_Table[5,118,0]:=-225242634;
   		 PHT_Table[5,118,1]:=57493;
   		 PHT_Table[0,119,0]:=2028716499;
   		 PHT_Table[0,119,1]:=61929;
   		 PHT_Table[1,119,0]:=-1385445386;
   		 PHT_Table[1,119,1]:=1249;
   		 PHT_Table[2,119,0]:=-581597661;
   		 PHT_Table[2,119,1]:=62973;
   		 PHT_Table[3,119,0]:=-2060020651;
   		 PHT_Table[3,119,1]:=61724;
   		 PHT_Table[4,119,0]:=545119088;
   		 PHT_Table[4,119,1]:=62728;
   		 PHT_Table[5,119,0]:=-118627226;
   		 PHT_Table[5,119,1]:=63804;
   		 PHT_Table[0,120,0]:=158699555;
   		 PHT_Table[0,120,1]:=25495;
   		 PHT_Table[1,120,0]:=399224111;
   		 PHT_Table[1,120,1]:=57138;
   		 PHT_Table[2,120,0]:=-1147108559;
   		 PHT_Table[2,120,1]:=48153;
   		 PHT_Table[3,120,0]:=281948320;
   		 PHT_Table[3,120,1]:=25387;
   		 PHT_Table[4,120,0]:=-1566079316;
   		 PHT_Table[4,120,1]:=48293;
   		 PHT_Table[5,120,0]:=-1219978048;
   		 PHT_Table[5,120,1]:=50825;
   		 PHT_Table[0,121,0]:=1177160904;
   		 PHT_Table[0,121,1]:=30663;
   		 PHT_Table[1,121,0]:=-1569120096;
   		 PHT_Table[1,121,1]:=49502;
   		 PHT_Table[2,121,0]:=2109177668;
   		 PHT_Table[2,121,1]:=46639;
   		 PHT_Table[3,121,0]:=1767357367;
   		 PHT_Table[3,121,1]:=30577;
   		 PHT_Table[4,121,0]:=1383879135;
   		 PHT_Table[4,121,1]:=46745;
   		 PHT_Table[5,121,0]:=352740570;
   		 PHT_Table[5,121,1]:=60963;
   		 PHT_Table[0,122,0]:=-1321343587;
   		 PHT_Table[0,122,1]:=44938;
   		 PHT_Table[1,122,0]:=-299948101;
   		 PHT_Table[1,122,1]:=30048;
   		 PHT_Table[2,122,0]:=-1250041628;
   		 PHT_Table[2,122,1]:=55856;
   		 PHT_Table[3,122,0]:=-2121754499;
   		 PHT_Table[3,122,1]:=44880;
   		 PHT_Table[4,122,0]:=-2062387365;
   		 PHT_Table[4,122,1]:=56042;
   		 PHT_Table[5,122,0]:=-1811954858;
   		 PHT_Table[5,122,1]:=17877;
   		 PHT_Table[0,123,0]:=246407371;
   		 PHT_Table[0,123,1]:=16915;
   		 PHT_Table[1,123,0]:=444284867;
   		 PHT_Table[1,123,1]:=25557;
   		 PHT_Table[2,123,0]:=-759165993;
   		 PHT_Table[2,123,1]:=8679;
   		 PHT_Table[3,123,0]:=-377675584;
   		 PHT_Table[3,123,1]:=16946;
   		 PHT_Table[4,123,0]:=892538312;
   		 PHT_Table[4,123,1]:=8646;
   		 PHT_Table[5,123,0]:=-630134656;
   		 PHT_Table[5,123,1]:=33799;
   		 PHT_Table[0,124,0]:=379091875;
   		 PHT_Table[0,124,1]:=8320;
   		 PHT_Table[1,124,0]:=-1648209148;
   		 PHT_Table[1,124,1]:=12512;
   		 PHT_Table[2,124,0]:=-338595185;
   		 PHT_Table[2,124,1]:=4208;
   		 PHT_Table[3,124,0]:=1718856401;
   		 PHT_Table[3,124,1]:=8336;
   		 PHT_Table[4,124,0]:=-1691696266;
   		 PHT_Table[4,124,1]:=4192;
   		 PHT_Table[5,124,0]:=1286659230;
   		 PHT_Table[5,124,1]:=16395;
   		 PHT_Table[0,125,0]:=934567224;
   		 PHT_Table[0,125,1]:=58809;
   		 PHT_Table[1,125,0]:=416893561;
   		 PHT_Table[1,125,1]:=6797;
   		 PHT_Table[2,125,0]:=457341526;
   		 PHT_Table[2,125,1]:=65483;
   		 PHT_Table[3,125,0]:=-55632062;
   		 PHT_Table[3,125,1]:=58694;
   		 PHT_Table[4,125,0]:=-794424317;
   		 PHT_Table[4,125,1]:=65332;
   		 PHT_Table[5,125,0]:=1520639100;
   		 PHT_Table[5,125,1]:=53654;
   		 PHT_Table[0,126,0]:=-1260472950;
   		 PHT_Table[0,126,1]:=64985;
   		 PHT_Table[1,126,0]:=923122810;
   		 PHT_Table[1,126,1]:=3781;
   		 PHT_Table[2,126,0]:=-1621568775;
   		 PHT_Table[2,126,1]:=62447;
   		 PHT_Table[3,126,0]:=1531047256;
   		 PHT_Table[3,126,1]:=64810;
   		 PHT_Table[4,126,0]:=1882494632;
   		 PHT_Table[4,126,1]:=62236;
   		 PHT_Table[5,126,0]:=1876379033;
   		 PHT_Table[5,126,1]:=57690;
   		 PHT_Table[0,127,0]:=-1166977727;
   		 PHT_Table[0,127,1]:=49098;
   		 PHT_Table[1,127,0]:=763265977;
   		 PHT_Table[1,127,1]:=27920;
   		 PHT_Table[2,127,0]:=1301862702;
   		 PHT_Table[2,127,1]:=53768;
   		 PHT_Table[3,127,0]:=-1304638056;
   		 PHT_Table[3,127,1]:=48920;
   		 PHT_Table[4,127,0]:=1158126432;
   		 PHT_Table[4,127,1]:=53978;
   		 PHT_Table[5,127,0]:=-1247302375;
   		 PHT_Table[5,127,1]:=25949;
   		 PHT_Table[0,128,0]:=1226112241;
   		 PHT_Table[0,128,1]:=33074;
   		 PHT_Table[1,128,0]:=-766011656;
   		 PHT_Table[1,128,1]:=19626;
   		 PHT_Table[2,128,0]:=64498019;
   		 PHT_Table[2,128,1]:=52565;
   		 PHT_Table[3,128,0]:=471278808;
   		 PHT_Table[3,128,1]:=33279;
   		 PHT_Table[4,128,0]:=1444309457;
   		 PHT_Table[4,128,1]:=52632;
   		 PHT_Table[5,128,0]:=176092560;
   		 PHT_Table[5,128,1]:=6569;
   		 PHT_Table[0,129,0]:=-2090145614;
   		 PHT_Table[0,129,1]:=6240;
   		 PHT_Table[1,129,0]:=803010051;
   		 PHT_Table[1,129,1]:=5192;
   		 PHT_Table[2,129,0]:=-2078627665;
   		 PHT_Table[2,129,1]:=3108;
   		 PHT_Table[3,129,0]:=-1477512678;
   		 PHT_Table[3,129,1]:=6252;
   		 PHT_Table[4,129,0]:=-1601004885;
   		 PHT_Table[4,129,1]:=3112;
   		 PHT_Table[5,129,0]:=896817637;
   		 PHT_Table[5,129,1]:=12492;
   		 PHT_Table[0,130,0]:=1880047874;
   		 PHT_Table[0,130,1]:=9880;
   		 PHT_Table[1,130,0]:=-789191870;
   		 PHT_Table[1,130,1]:=13810;
   		 PHT_Table[2,130,0]:=-900048670;
   		 PHT_Table[2,130,1]:=4985;
   		 PHT_Table[3,130,0]:=163912538;
   		 PHT_Table[3,130,1]:=9867;
   		 PHT_Table[4,130,0]:=-1283233766;
   		 PHT_Table[4,130,1]:=4970;
   		 PHT_Table[5,130,0]:=-1968373396;
   		 PHT_Table[5,130,1]:=19512;
   		 PHT_Table[0,131,0]:=1203444794;
   		 PHT_Table[0,131,1]:=49953;
   		 PHT_Table[1,131,0]:=-936597189;
   		 PHT_Table[1,131,1]:=12159;
   		 PHT_Table[2,131,0]:=-786947404;
   		 PHT_Table[2,131,1]:=60594;
   		 PHT_Table[3,131,0]:=-177601512;
   		 PHT_Table[3,131,1]:=50125;
   		 PHT_Table[4,131,0]:=1663394841;
   		 PHT_Table[4,131,1]:=60510;
   		 PHT_Table[5,131,0]:=-804381424;
   		 PHT_Table[5,131,1]:=40366;
   		 PHT_Table[0,132,0]:=-1422696950;
   		 PHT_Table[0,132,1]:=48846;
   		 PHT_Table[1,132,0]:=-1123270063;
   		 PHT_Table[1,132,1]:=57623;
   		 PHT_Table[2,132,0]:=-819387577;
   		 PHT_Table[2,132,1]:=24454;
   		 PHT_Table[3,132,0]:=771520297;
   		 PHT_Table[3,132,1]:=48785;
   		 PHT_Table[4,132,0]:=1236915058;
   		 PHT_Table[4,132,1]:=24537;
   		 PHT_Table[5,132,0]:=-1808857657;
   		 PHT_Table[5,132,1]:=26584;
   		 PHT_Table[0,133,0]:=1216736259;
   		 PHT_Table[0,133,1]:=13780;
   		 PHT_Table[1,133,0]:=-1207820445;
   		 PHT_Table[1,133,1]:=41611;
   		 PHT_Table[2,133,0]:=-1351125869;
   		 PHT_Table[2,133,1]:=38856;
   		 PHT_Table[3,133,0]:=-2144691337;
   		 PHT_Table[3,133,1]:=13635;
   		 PHT_Table[4,133,0]:=1733254167;
   		 PHT_Table[4,133,1]:=38751;
   		 PHT_Table[5,133,0]:=-814314406;
   		 PHT_Table[5,133,1]:=27172;
   		 PHT_Table[0,134,0]:=-797921324;
   		 PHT_Table[0,134,1]:=34838;
   		 PHT_Table[1,134,0]:=-1365768943;
   		 PHT_Table[1,134,1]:=52373;
   		 PHT_Table[2,134,0]:=-40484241;
   		 PHT_Table[2,134,1]:=17607;
   		 PHT_Table[3,134,0]:=395131286;
   		 PHT_Table[3,134,1]:=34898;
   		 PHT_Table[4,134,0]:=976181075;
   		 PHT_Table[4,134,1]:=17539;
   		 PHT_Table[5,134,0]:=953838308;
   		 PHT_Table[5,134,1]:=2920;
   		 PHT_Table[0,135,0]:=-131524244;
   		 PHT_Table[0,135,1]:=11960;
   		 PHT_Table[1,135,0]:=1011396931;
   		 PHT_Table[1,135,1]:=14794;
   		 PHT_Table[2,135,0]:=-1230648953;
   		 PHT_Table[2,135,1]:=5989;
   		 PHT_Table[3,135,0]:=-1650475867;
   		 PHT_Table[3,135,1]:=11951;
   		 PHT_Table[4,135,0]:=-754704758;
   		 PHT_Table[4,135,1]:=6002;
   		 PHT_Table[5,135,0]:=-1719585082;
   		 PHT_Table[5,135,1]:=23676;
   		 PHT_Table[0,136,0]:=1625053883;
   		 PHT_Table[0,136,1]:=37754;
   		 PHT_Table[1,136,0]:=718449457;
   		 PHT_Table[1,136,1]:=22484;
   		 PHT_Table[2,136,0]:=-465240197;
   		 PHT_Table[2,136,1]:=50282;
   		 PHT_Table[3,136,0]:=171449924;
   		 PHT_Table[3,136,1]:=37822;
   		 PHT_Table[4,136,0]:=-1906043442;
   		 PHT_Table[4,136,1]:=50350;
   		 PHT_Table[5,136,0]:=1848496248;
   		 PHT_Table[5,136,1]:=15664;
   		 PHT_Table[0,137,0]:=1916166653;
   		 PHT_Table[0,137,1]:=21839;
   		 PHT_Table[1,137,0]:=73394799;
   		 PHT_Table[1,137,1]:=62128;
   		 PHT_Table[2,137,0]:=-1994399207;
   		 PHT_Table[2,137,1]:=42840;
   		 PHT_Table[3,137,0]:=717192735;
   		 PHT_Table[3,137,1]:=21992;
   		 PHT_Table[4,137,0]:=-785317235;
   		 PHT_Table[4,137,1]:=43007;
   		 PHT_Table[5,137,0]:=465433571;
   		 PHT_Table[5,137,1]:=43577;
   		 PHT_Table[0,138,0]:=-1516454207;
   		 PHT_Table[0,138,1]:=64733;
   		 PHT_Table[1,138,0]:=-1485341294;
   		 PHT_Table[1,138,1]:=33474;
   		 PHT_Table[2,138,0]:=501819536;
   		 PHT_Table[2,138,1]:=32353;
   		 PHT_Table[3,138,0]:=-998156311;
   		 PHT_Table[3,138,1]:=64675;
   		 PHT_Table[4,138,0]:=2089475770;
   		 PHT_Table[4,138,1]:=32287;
   		 PHT_Table[5,138,0]:=1314909511;
   		 PHT_Table[5,138,1]:=58335;
   		 PHT_Table[0,139,0]:=-1688374310;
